C07281=1024.683,249.663,375.883,169.871,47.896,159.167
C07282=1024.672,249.258,375.931,169.865,47.901,159.167
C07283=1024.662,248.853,375.977,169.859,47.906,159.167
C07284=1024.652,248.448,376.024,169.852,47.911,159.167
C07285=1024.641,248.044,376.071,169.847,47.915,159.168
C07286=1024.635,247.795,376.099,169.843,47.919,159.168
C07287=1024.628,247.547,376.128,169.839,47.921,159.168
C07288=1024.622,247.299,376.157,169.835,47.924,159.168
C07289=1024.616,247.050,376.185,169.832,47.927,159.168
C07290=1024.609,246.802,376.213,169.827,47.930,159.168
C07291=1024.603,246.554,376.242,169.824,47.933,159.168
C07292=1024.597,246.305,376.271,169.821,47.935,159.168
C07293=1024.590,246.057,376.298,169.817,47.939,159.169
C07294=1024.584,245.809,376.327,169.813,47.941,159.169
C07295=1024.578,245.560,376.356,169.809,47.944,159.169
C07296=1024.572,245.312,376.385,169.806,47.947,159.169
C07297=1024.565,245.064,376.413,169.802,47.950,159.169
C07298=1024.560,244.816,376.441,169.799,47.953,159.169
C07299=1024.554,244.567,376.470,169.794,47.956,159.169
C07300=1024.547,244.320,376.498,169.791,47.959,159.170
C07301=1024.541,244.071,376.526,169.787,47.962,159.170
C07302=1024.535,243.823,376.555,169.784,47.965,159.170
C07303=1024.528,243.574,376.583,169.779,47.968,159.170
C07304=1024.522,243.325,376.611,169.776,47.971,159.170
C07305=1024.515,243.078,376.640,169.772,47.974,159.170
C07306=1024.508,242.829,376.668,169.769,47.977,159.170
C07307=1024.502,242.580,376.696,169.765,47.980,159.171
C07308=1024.495,242.333,376.724,169.762,47.983,159.171
C07309=1024.490,242.085,376.752,169.758,47.987,159.171
C07310=1024.483,241.836,376.780,169.754,47.989,159.171
C07311=1024.477,241.588,376.808,169.750,47.993,159.171
C07312=1024.471,241.339,376.836,169.747,47.996,159.171
C07313=1024.464,241.091,376.865,169.743,47.999,159.172
C07314=1024.458,240.842,376.893,169.740,48.002,159.172
C07315=1024.451,240.594,376.921,169.735,48.005,159.172
C07316=1024.445,240.345,376.949,169.732,48.008,159.172
C07317=1024.438,240.097,376.977,169.728,48.011,159.172
C07318=1024.432,239.850,377.005,169.725,48.015,159.173
C07319=1024.426,239.601,377.033,169.721,48.017,159.173
C07320=1024.419,239.352,377.061,169.718,48.020,159.173
C07321=1024.413,239.104,377.089,169.714,48.024,159.173
C07322=1024.406,238.856,377.116,169.711,48.027,159.173
C07323=1024.399,238.607,377.144,169.707,48.030,159.173
C07324=1024.394,238.359,377.172,169.703,48.033,159.174
C07325=1024.387,238.111,377.200,169.699,48.037,159.174
C07326=1024.381,237.862,377.227,169.696,48.040,159.174
C07327=1024.374,237.614,377.255,169.692,48.043,159.174
C07328=1024.367,237.365,377.283,169.688,48.047,159.174
C07329=1024.361,237.117,377.311,169.685,48.050,159.175
C07330=1024.355,236.869,377.339,169.681,48.053,159.175
C07331=1024.349,236.620,377.366,169.678,48.056,159.175
C07332=1024.342,236.372,377.394,169.674,48.060,159.175
C07333=1024.336,236.123,377.421,169.671,48.063,159.176
C07334=1024.329,235.874,377.449,169.667,48.066,159.176
C07335=1024.323,235.627,377.476,169.664,48.070,159.176
C07336=1024.316,235.378,377.504,169.660,48.073,159.176
C07337=1024.309,235.130,377.532,169.657,48.076,159.176
C07338=1024.299,234.719,377.577,169.650,48.082,159.177
C07339=1024.288,234.308,377.623,169.645,48.087,159.177
C07340=1024.277,233.897,377.668,169.638,48.093,159.177
C07341=1024.267,233.486,377.714,169.633,48.098,159.178
C07342=1024.260,233.238,377.741,169.629,48.101,159.178
C07343=1024.255,232.988,377.769,169.626,48.104,159.178
C07344=1024.248,232.740,377.797,169.622,48.108,159.179
C07345=1024.242,232.492,377.824,169.619,48.112,159.179
C07346=1024.235,232.244,377.852,169.615,48.115,159.179
C07347=1024.229,231.995,377.879,169.612,48.118,159.179
C07348=1024.223,231.747,377.906,169.608,48.122,159.179
C07349=1024.216,231.499,377.934,169.604,48.125,159.180
C07350=1024.210,231.249,377.961,169.600,48.128,159.180
C07351=1024.204,231.002,377.988,169.598,48.132,159.180
C07352=1024.197,230.753,378.016,169.594,48.135,159.180
C07353=1024.190,230.505,378.044,169.591,48.138,159.181
C07354=1024.185,230.256,378.071,169.586,48.142,159.181
C07355=1024.178,230.008,378.098,169.583,48.145,159.181
C07356=1024.172,229.759,378.125,169.580,48.149,159.181
C07357=1024.165,229.511,378.153,169.577,48.152,159.182
C07358=1024.159,229.262,378.180,169.573,48.156,159.182
C07359=1024.152,229.014,378.207,169.569,48.159,159.182
C07360=1024.146,228.766,378.235,169.566,48.163,159.182
C07361=1024.140,228.517,378.262,169.562,48.166,159.183
C07362=1024.133,228.268,378.289,169.559,48.169,159.183
C07363=1024.127,228.020,378.316,169.555,48.173,159.183
C07364=1024.120,227.772,378.343,169.552,48.177,159.183
C07365=1024.114,227.523,378.370,169.548,48.180,159.184
C07366=1024.108,227.275,378.398,169.545,48.184,159.184
C07367=1024.101,227.026,378.425,169.541,48.187,159.184
C07368=1024.095,226.778,378.451,169.538,48.190,159.184
C07369=1024.088,226.530,378.478,169.534,48.194,159.185
C07370=1024.082,226.281,378.505,169.531,48.198,159.185
C07371=1024.076,226.033,378.533,169.527,48.202,159.185
C07372=1024.068,225.784,378.559,169.524,48.205,159.186
C07373=1024.063,225.536,378.586,169.520,48.209,159.186
C07374=1024.056,225.287,378.614,169.516,48.212,159.186
C07375=1024.049,225.039,378.640,169.514,48.216,159.187
C07376=1024.043,224.790,378.667,169.510,48.220,159.187
C07377=1024.037,224.541,378.694,169.507,48.223,159.187
C07378=1024.031,224.293,378.721,169.503,48.227,159.187
C07379=1024.024,224.045,378.747,169.500,48.231,159.188
C07380=1024.018,223.796,378.774,169.496,48.234,159.188
C07381=1024.011,223.547,378.801,169.493,48.238,159.188
C07382=1024.004,223.299,378.828,169.489,48.241,159.189
C07383=1023.998,223.051,378.855,169.486,48.245,159.189
C07384=1023.992,222.802,378.882,169.482,48.248,159.189
C07385=1023.985,222.554,378.908,169.479,48.253,159.190
C07386=1023.979,222.305,378.936,169.476,48.256,159.190
C07387=1023.973,222.057,378.962,169.472,48.260,159.190
C07388=1023.966,221.808,378.989,169.469,48.263,159.190
C07389=1023.960,221.560,379.015,169.465,48.267,159.191
C07390=1023.954,221.311,379.042,169.462,48.271,159.191
C07391=1023.947,221.063,379.069,169.458,48.274,159.191
C07392=1023.940,220.814,379.096,169.456,48.278,159.192
C07393=1023.935,220.566,379.123,169.451,48.282,159.192
C07394=1023.924,220.147,379.168,169.446,48.288,159.192
C07395=1023.913,219.728,379.213,169.441,48.294,159.193
C07396=1023.902,219.309,379.258,169.434,48.301,159.194
C07397=1023.892,218.890,379.302,169.429,48.307,159.194
C07398=1023.885,218.641,379.329,169.426,48.311,159.195
C07399=1023.879,218.393,379.355,169.422,48.314,159.195
C07400=1023.872,218.144,379.382,169.419,48.318,159.195
C07401=1023.866,217.896,379.408,169.415,48.322,159.195
C07402=1023.859,217.648,379.434,169.412,48.326,159.196
C07403=1023.852,217.399,379.461,169.408,48.329,159.196
C07404=1023.847,217.151,379.487,169.406,48.333,159.196
C07405=1023.839,216.902,379.514,169.402,48.337,159.197
C07406=1023.834,216.654,379.540,169.398,48.342,159.197
C07407=1023.827,216.405,379.567,169.395,48.345,159.198
C07408=1023.820,216.157,379.593,169.392,48.349,159.198
C07409=1023.814,215.909,379.620,169.389,48.353,159.198
C07410=1023.808,215.659,379.645,169.385,48.357,159.199
C07411=1023.801,215.411,379.671,169.382,48.361,159.199
C07412=1023.795,215.162,379.698,169.378,48.365,159.199
C07413=1023.788,214.914,379.724,169.375,48.369,159.200
C07414=1023.782,214.666,379.751,169.372,48.373,159.200
C07415=1023.775,214.417,379.777,169.368,48.377,159.200
C07416=1023.769,214.168,379.803,169.365,48.380,159.201
C07417=1023.763,213.919,379.830,169.362,48.384,159.201
C07418=1023.756,213.671,379.856,169.359,48.388,159.201
C07419=1023.750,213.423,379.882,169.355,48.392,159.202
C07420=1023.743,213.174,379.909,169.351,48.396,159.202
C07421=1023.737,212.925,379.934,169.349,48.400,159.203
C07422=1023.731,212.677,379.960,169.345,48.404,159.203
C07423=1023.724,212.428,379.987,169.342,48.408,159.203
C07424=1023.718,212.180,380.013,169.338,48.412,159.204
C07425=1023.712,211.931,380.039,169.336,48.416,159.204
C07426=1023.705,211.682,380.066,169.332,48.420,159.204
C07427=1023.699,211.434,380.092,169.329,48.424,159.205
C07428=1023.693,211.185,380.118,169.326,48.428,159.205
C07429=1023.686,210.937,380.144,169.321,48.431,159.205
C07430=1023.679,210.689,380.170,169.319,48.435,159.206
C07431=1023.674,210.440,380.196,169.315,48.439,159.206
C07432=1023.667,210.192,380.222,169.312,48.443,159.207
C07433=1023.660,209.943,380.249,169.309,48.448,159.207
C07434=1023.654,209.694,380.274,169.306,48.452,159.208
C07435=1023.648,209.446,380.300,169.303,48.456,159.208
C07436=1023.642,209.196,380.326,169.299,48.460,159.208
C07437=1023.635,208.948,380.352,169.296,48.464,159.209
C07438=1023.629,208.700,380.378,169.292,48.468,159.209
C07439=1023.622,208.452,380.404,169.290,48.472,159.209
C07440=1023.615,208.203,380.430,169.286,48.476,159.210
C07441=1023.609,207.954,380.456,169.282,48.480,159.210
C07442=1023.603,207.706,380.482,169.279,48.484,159.211
C07443=1023.597,207.457,380.508,169.276,48.488,159.211
C07444=1023.590,207.208,380.534,169.273,48.492,159.212
C07445=1023.584,206.960,380.559,169.270,48.496,159.212
C07446=1023.577,206.712,380.585,169.266,48.501,159.212
C07447=1023.571,206.463,380.611,169.263,48.504,159.213
C07448=1023.564,206.214,380.636,169.260,48.509,159.213
C07449=1023.558,205.966,380.662,169.257,48.513,159.214
C07450=1023.547,205.550,380.705,169.251,48.520,159.214
C07451=1023.536,205.133,380.749,169.246,48.527,159.215
C07452=1023.525,204.716,380.791,169.240,48.534,159.216
C07453=1023.515,204.300,380.834,169.236,48.541,159.216
C07454=1023.491,203.269,380.934,168.819,48.442,159.136
C07455=1023.486,203.020,380.959,168.815,48.447,159.136
C07456=1023.480,202.772,380.983,168.811,48.452,159.136
C07457=1023.474,202.523,381.007,168.806,48.457,159.137
C07458=1023.469,202.274,381.031,168.802,48.463,159.137
C07459=1023.464,202.025,381.055,168.798,48.468,159.138
C07460=1023.458,201.776,381.079,168.794,48.472,159.138
C07461=1023.452,201.528,381.103,168.790,48.478,159.139
C07462=1023.446,201.279,381.127,168.786,48.483,159.139
C07463=1023.441,201.030,381.152,168.781,48.488,159.140
C07464=1023.436,200.781,381.175,168.778,48.493,159.140
C07465=1023.429,200.532,381.199,168.773,48.498,159.141
C07466=1023.424,200.284,381.223,168.769,48.503,159.141
C07467=1023.419,200.035,381.248,168.764,48.509,159.141
C07468=1023.413,199.786,381.272,168.761,48.513,159.142
C07469=1023.407,199.537,381.295,168.757,48.518,159.142
C07470=1023.402,199.288,381.319,168.753,48.524,159.143
C07471=1023.396,199.039,381.342,168.748,48.529,159.143
C07472=1023.390,198.791,381.366,168.744,48.534,159.144
C07473=1023.385,198.542,381.390,168.740,48.539,159.144
C07474=1023.378,198.293,381.414,168.736,48.545,159.145
C07475=1023.372,198.045,381.437,168.732,48.550,159.145
C07476=1023.367,197.795,381.461,168.727,48.555,159.146
C07477=1023.361,197.547,381.485,168.724,48.561,159.146
C07478=1023.356,197.298,381.508,168.720,48.566,159.147
C07479=1023.350,197.049,381.532,168.715,48.571,159.147
C07480=1023.344,196.800,381.555,168.711,48.576,159.148
C07481=1023.339,196.551,381.579,168.708,48.582,159.148
C07482=1023.333,196.303,381.602,168.703,48.587,159.149
C07483=1023.328,196.054,381.626,168.699,48.592,159.149
C07484=1023.322,195.805,381.649,168.695,48.598,159.150
C07485=1023.316,195.557,381.673,168.692,48.602,159.150
C07486=1023.310,195.307,381.697,168.687,48.608,159.151
C07487=1023.305,195.058,381.720,168.683,48.613,159.151
C07488=1023.299,194.810,381.744,168.679,48.619,159.152
C07489=1023.294,194.560,381.767,168.675,48.623,159.152
C07490=1023.288,194.312,381.791,168.671,48.628,159.152
C07491=1023.283,194.063,381.814,168.667,48.634,159.153
C07492=1023.277,193.814,381.837,168.663,48.639,159.154
C07493=1023.271,193.566,381.861,168.659,48.644,159.154
C07494=1023.266,193.317,381.884,168.655,48.650,159.155
C07495=1023.260,193.068,381.908,168.651,48.655,159.155
C07496=1023.254,192.819,381.931,168.647,48.660,159.155
C07497=1023.249,192.570,381.955,168.643,48.666,159.156
C07498=1023.243,192.321,381.978,168.640,48.671,159.157
C07499=1023.238,192.073,382.002,168.635,48.676,159.157
C07500=1023.232,191.824,382.025,168.631,48.682,159.158
C07501=1023.227,191.575,382.048,168.628,48.686,159.158
C07502=1023.221,191.326,382.072,168.623,48.692,159.158
C07503=1023.215,191.077,382.095,168.619,48.697,159.159
C07504=1023.210,190.829,382.118,168.616,48.702,159.160
C07505=1023.205,190.579,382.141,168.611,48.707,159.160
C07506=1023.199,190.331,382.165,168.607,48.713,159.161
C07507=1023.193,190.082,382.188,168.604,48.718,159.161
C07508=1023.188,189.833,382.212,168.600,48.724,159.162
C07509=1023.182,189.584,382.235,168.595,48.729,159.162
C07510=1023.177,189.336,382.259,168.592,48.734,159.163
C07511=1023.171,189.087,382.282,168.588,48.740,159.163
C07512=1023.166,188.838,382.305,168.584,48.744,159.164
C07513=1023.161,188.588,382.328,168.580,48.750,159.164
C07514=1023.155,188.340,382.351,168.576,48.755,159.165
C07515=1023.148,188.058,382.378,168.572,48.761,159.165
C07516=1023.142,187.776,382.404,168.568,48.767,159.166
C07517=1023.136,187.494,382.430,168.563,48.773,159.166
C07518=1023.131,187.212,382.457,168.559,48.779,159.167
C07519=1023.125,186.963,382.479,168.555,48.784,159.167
C07520=1023.119,186.714,382.502,168.551,48.790,159.168
C07521=1023.114,186.465,382.526,168.547,48.795,159.168
C07522=1023.108,186.216,382.549,168.543,48.800,159.169
C07523=1023.102,185.967,382.573,168.539,48.806,159.169
C07524=1023.097,185.718,382.596,168.536,48.810,159.170
C07525=1023.092,185.469,382.619,168.532,48.816,159.171
C07526=1023.087,185.221,382.642,168.529,48.821,159.171
C07527=1023.082,184.972,382.665,168.524,48.826,159.171
C07528=1023.076,184.723,382.688,168.521,48.832,159.172
C07529=1023.070,184.474,382.711,168.517,48.837,159.173
C07530=1023.065,184.225,382.735,168.513,48.842,159.173
C07531=1023.059,183.976,382.758,168.509,48.848,159.174
C07532=1023.054,183.728,382.780,168.506,48.853,159.174
C07533=1023.049,183.479,382.804,168.502,48.858,159.175
C07534=1023.044,183.230,382.827,168.498,48.863,159.175
C07535=1023.038,182.981,382.850,168.494,48.868,159.176
C07536=1023.033,182.731,382.872,168.491,48.874,159.176
C07537=1023.027,182.482,382.895,168.487,48.879,159.177
C07538=1023.022,182.234,382.918,168.484,48.885,159.177
C07539=1023.017,181.985,382.941,168.479,48.890,159.178
C07540=1023.011,181.735,382.963,168.475,48.896,159.178
C07541=1023.005,181.487,382.985,168.472,48.901,159.179
C07542=1022.999,181.238,383.008,168.468,48.907,159.180
C07543=1022.993,180.988,383.031,168.464,48.912,159.180
C07544=1022.988,180.741,383.053,168.461,48.918,159.181
C07545=1022.982,180.491,383.075,168.457,48.924,159.181
C07546=1022.976,180.242,383.098,168.453,48.929,159.182
C07547=1022.971,179.993,383.121,168.449,48.934,159.182
C07548=1022.965,179.744,383.142,168.445,48.940,159.183
C07549=1022.959,179.495,383.165,168.442,48.946,159.184
C07550=1022.954,179.246,383.187,168.438,48.951,159.184
C07551=1022.948,178.998,383.210,168.435,48.957,159.185
C07552=1022.942,178.748,383.232,168.431,48.962,159.185
C07553=1022.936,178.499,383.255,168.426,48.968,159.186
C07554=1022.931,178.251,383.276,168.423,48.973,159.186
C07555=1022.925,178.002,383.299,168.419,48.979,159.187
C07556=1022.920,177.752,383.321,168.416,48.985,159.188
C07557=1022.914,177.504,383.344,168.412,48.990,159.188
C07558=1022.908,177.255,383.365,168.409,48.995,159.189
C07559=1022.903,177.006,383.388,168.405,49.001,159.189
C07560=1022.897,176.757,383.411,168.401,49.006,159.190
C07561=1022.891,176.508,383.433,168.397,49.012,159.190
C07562=1022.886,176.259,383.455,168.393,49.018,159.191
C07563=1022.880,176.010,383.478,168.390,49.023,159.192
C07564=1022.874,175.761,383.499,168.386,49.029,159.192
C07565=1022.869,175.513,383.522,168.383,49.034,159.193
C07566=1022.863,175.263,383.544,168.379,49.040,159.193
C07567=1022.858,175.014,383.566,168.376,49.046,159.194
C07568=1022.852,174.766,383.588,168.371,49.051,159.194
C07569=1022.847,174.516,383.611,168.368,49.056,159.195
C07570=1022.841,174.268,383.634,168.364,49.062,159.195
C07571=1022.835,174.019,383.655,168.361,49.068,159.196
C07572=1022.830,173.770,383.677,168.357,49.073,159.197
C07573=1022.824,173.521,383.700,168.354,49.079,159.197
C07574=1022.819,173.272,383.721,168.350,49.084,159.198
C07575=1022.813,173.023,383.743,168.346,49.089,159.198
C07576=1022.808,172.774,383.766,168.342,49.095,159.199
C07577=1022.802,172.525,383.788,168.339,49.101,159.200
C07578=1022.797,172.276,383.810,168.335,49.107,159.200
C07579=1022.791,171.993,383.836,168.331,49.113,159.201
C07580=1022.784,171.711,383.860,168.328,49.119,159.201
C07581=1022.778,171.428,383.886,168.324,49.125,159.202
C07582=1022.771,171.146,383.911,168.320,49.132,159.203
C07583=1022.766,170.897,383.933,168.315,49.137,159.203
C07584=1022.760,170.648,383.954,168.312,49.142,159.204
C07585=1022.755,170.399,383.976,168.308,49.148,159.204
C07586=1022.750,170.150,383.999,168.305,49.154,159.205
C07587=1022.744,169.901,384.021,168.301,49.159,159.206
C07588=1022.739,169.652,384.042,168.298,49.165,159.206
C07589=1022.734,169.403,384.065,168.295,49.170,159.207
C07590=1022.728,169.154,384.086,168.291,49.176,159.207
C07591=1022.722,168.905,384.109,168.288,49.181,159.208
C07592=1022.717,168.657,384.131,168.284,49.187,159.208
C07593=1022.711,168.407,384.152,168.281,49.192,159.209
C07594=1022.706,168.158,384.175,168.277,49.197,159.210
C07595=1022.701,167.909,384.197,168.273,49.203,159.210
C07596=1022.695,167.660,384.218,168.270,49.209,159.211
C07597=1022.690,167.412,384.241,168.266,49.215,159.211
C07598=1022.684,167.162,384.263,168.263,49.220,159.212
C07599=1022.679,166.914,384.284,168.260,49.225,159.213
C07600=1022.674,166.665,384.306,168.256,49.231,159.213
C07601=1022.668,166.415,384.328,168.253,49.237,159.214
C07602=1022.663,166.167,384.350,168.250,49.242,159.214
C07603=1022.657,165.917,384.372,168.246,49.248,159.215
C07604=1022.653,165.669,384.394,168.243,49.253,159.216
C07605=1022.646,165.419,384.415,168.240,49.259,159.216
C07606=1022.642,165.170,384.437,168.235,49.264,159.217
C07607=1022.636,164.922,384.460,168.232,49.270,159.217
C07608=1022.630,164.673,384.481,168.228,49.276,159.218
C07609=1022.625,164.424,384.504,168.225,49.280,159.218
C07610=1022.620,164.175,384.525,168.222,49.286,159.219
C07611=1022.615,163.926,384.547,168.218,49.292,159.220
C07612=1022.609,163.677,384.569,168.215,49.298,159.220
C07613=1022.604,163.428,384.591,168.211,49.303,159.221
C07614=1022.598,163.179,384.612,168.209,49.308,159.221
C07615=1022.593,162.930,384.634,168.204,49.314,159.222
C07616=1022.588,162.681,384.656,168.201,49.319,159.222
C07617=1022.582,162.432,384.678,168.198,49.325,159.223
C07618=1022.578,162.183,384.700,168.194,49.331,159.224
C07619=1022.572,161.934,384.722,168.191,49.336,159.224
C07620=1022.567,161.684,384.743,168.188,49.341,159.225
C07621=1022.562,161.436,384.764,168.184,49.347,159.225
C07622=1022.556,161.186,384.786,168.181,49.353,159.226
C07623=1022.551,160.938,384.808,168.178,49.358,159.227
C07624=1022.546,160.689,384.830,168.175,49.363,159.227
C07625=1022.540,160.440,384.851,168.171,49.369,159.228
C07626=1022.535,160.191,384.873,168.168,49.375,159.228
C07627=1022.530,159.942,384.895,168.164,49.380,159.229
C07628=1022.524,159.693,384.917,168.161,49.385,159.230
C07629=1022.519,159.444,384.939,168.157,49.391,159.230
C07630=1022.515,159.194,384.960,168.154,49.397,159.231
C07631=1022.509,158.945,384.981,168.151,49.402,159.231
C07632=1022.503,158.697,385.003,168.147,49.408,159.232
C07633=1022.498,158.448,385.024,168.144,49.413,159.233
C07634=1022.492,158.198,385.045,168.141,49.419,159.233
C07635=1022.487,157.950,385.067,168.137,49.425,159.234
C07636=1022.482,157.700,385.087,168.134,49.431,159.234
C07637=1022.475,157.451,385.109,168.131,49.436,159.235
C07638=1022.470,157.203,385.130,168.127,49.442,159.236
C07639=1022.465,156.953,385.151,168.124,49.448,159.236
C07640=1022.459,156.704,385.173,168.121,49.453,159.237
C07641=1022.454,156.456,385.194,168.117,49.459,159.238
C07642=1022.448,156.207,385.215,168.114,49.465,159.238
C07643=1022.442,155.924,385.239,168.110,49.471,159.239
C07644=1022.436,155.640,385.263,168.106,49.477,159.240
C07645=1022.429,155.358,385.287,168.103,49.484,159.240
C07646=1022.423,155.075,385.311,168.099,49.491,159.241
C07647=1022.418,154.826,385.332,168.096,49.496,159.242
C07648=1022.413,154.577,385.354,168.092,49.502,159.242
C07649=1022.407,154.327,385.375,168.089,49.507,159.243
C07650=1022.402,154.079,385.396,168.086,49.513,159.243
C07651=1022.396,153.830,385.417,168.082,49.519,159.244
C07652=1022.390,153.580,385.438,168.079,49.525,159.245
C07653=1022.385,153.331,385.459,168.076,49.530,159.245
C07654=1022.380,153.083,385.481,168.073,49.536,159.246
C07655=1022.375,152.833,385.501,168.069,49.542,159.247
C07656=1022.369,152.584,385.522,168.066,49.547,159.247
C07657=1022.363,152.335,385.543,168.063,49.553,159.248
C07658=1022.358,152.086,385.564,168.059,49.559,159.249
C07659=1022.353,151.837,385.585,168.056,49.565,159.249
C07660=1022.347,151.588,385.606,168.053,49.570,159.250
C07661=1022.341,151.338,385.627,168.049,49.576,159.250
C07662=1022.336,151.090,385.648,168.046,49.582,159.251
C07663=1022.331,150.841,385.669,168.043,49.588,159.252
C07664=1022.325,150.592,385.689,168.040,49.593,159.252
C07665=1022.319,150.343,385.711,168.036,49.599,159.253
C07666=1022.314,150.093,385.731,168.034,49.605,159.254
C07667=1022.309,149.844,385.752,168.031,49.611,159.254
C07668=1022.303,149.596,385.773,168.028,49.616,159.255
C07669=1022.298,149.347,385.794,168.024,49.622,159.256
C07670=1022.292,149.097,385.815,168.021,49.628,159.256
C07671=1022.286,148.848,385.836,168.018,49.633,159.257
C07672=1022.281,148.599,385.856,168.014,49.639,159.257
C07673=1022.276,148.350,385.877,168.011,49.645,159.258
C07674=1022.271,148.101,385.897,168.008,49.651,159.259
C07675=1022.265,147.852,385.919,168.005,49.656,159.259
C07676=1022.259,147.603,385.940,168.001,49.662,159.260
C07677=1022.254,147.353,385.960,167.998,49.668,159.261
C07678=1022.249,147.104,385.981,167.995,49.674,159.261
C07679=1022.243,146.856,386.002,167.992,49.679,159.262
C07680=1022.238,146.607,386.023,167.988,49.685,159.263
C07681=1022.232,146.358,386.043,167.985,49.691,159.263
C07682=1022.226,146.108,386.063,167.982,49.697,159.264
C07683=1022.221,145.859,386.084,167.979,49.702,159.265
C07684=1022.216,145.610,386.105,167.975,49.708,159.265
C07685=1022.210,145.361,386.125,167.972,49.714,159.266
C07686=1022.205,145.112,386.146,167.970,49.720,159.267
C07687=1022.199,144.863,386.166,167.967,49.726,159.267
C07688=1022.194,144.614,386.187,167.963,49.732,159.268
C07689=1022.188,144.364,386.208,167.960,49.738,159.268
C07690=1022.182,144.115,386.228,167.957,49.743,159.269
C07691=1022.176,143.867,386.248,167.954,49.749,159.270
C07692=1022.171,143.617,386.269,167.950,49.755,159.270
C07693=1022.166,143.368,386.289,167.947,49.761,159.271
C07694=1022.161,143.119,386.310,167.944,49.766,159.272
C07695=1022.155,142.870,386.330,167.941,49.772,159.272
C07696=1022.149,142.621,386.351,167.937,49.778,159.273
C07697=1022.144,142.372,386.371,167.935,49.784,159.274
C07698=1022.138,142.123,386.391,167.932,49.790,159.274
C07699=1022.133,141.874,386.412,167.929,49.796,159.275
C07700=1022.127,141.624,386.433,167.926,49.801,159.276
C07701=1022.122,141.375,386.453,167.922,49.807,159.276
C07702=1022.116,141.126,386.473,167.919,49.813,159.277
C07703=1022.111,140.877,386.494,167.916,49.819,159.278
C07704=1022.105,140.628,386.514,167.913,49.825,159.278
C07705=1022.100,140.379,386.535,167.909,49.831,159.279
C07706=1022.094,140.130,386.554,167.906,49.836,159.280
C07707=1022.089,139.893,386.574,167.904,49.842,159.280
C07708=1022.084,139.654,386.593,167.901,49.848,159.281
C07709=1022.079,139.416,386.613,167.898,49.853,159.282
C07710=1022.074,139.177,386.632,167.894,49.858,159.282
C07711=1022.069,138.940,386.652,167.891,49.864,159.283
C07712=1022.064,138.701,386.671,167.890,49.869,159.283
C07713=1022.058,138.463,386.691,167.887,49.875,159.284
C07714=1022.053,138.225,386.709,167.884,49.881,159.285
C07715=1022.047,137.919,386.735,167.879,49.888,159.285
C07716=1022.040,137.615,386.760,167.876,49.895,159.286
C07717=1022.033,137.310,386.784,167.871,49.902,159.287
C07718=1022.026,137.004,386.809,167.868,49.910,159.288
C07719=1022.020,136.755,386.829,167.865,49.915,159.289
C07720=1022.015,136.506,386.849,167.862,49.921,159.289
C07721=1022.009,136.257,386.869,167.859,49.927,159.290
C07722=1022.004,136.007,386.889,167.855,49.933,159.290
C07723=1021.998,135.759,386.909,167.853,49.938,159.291
C07724=1021.993,135.509,386.929,167.850,49.944,159.292
C07725=1021.987,135.260,386.949,167.847,49.950,159.293
C07726=1021.982,135.012,386.969,167.844,49.956,159.293
C07727=1021.977,134.762,386.988,167.840,49.962,159.294
C07728=1021.971,134.513,387.009,167.837,49.968,159.295
C07729=1021.965,134.264,387.029,167.834,49.974,159.295
C07730=1021.960,134.015,387.049,167.831,49.979,159.296
C07731=1021.954,133.766,387.069,167.829,49.985,159.296
C07732=1021.949,133.517,387.089,167.825,49.992,159.297
C07733=1021.943,133.267,387.108,167.822,49.997,159.298
C07734=1021.938,133.018,387.129,167.819,50.003,159.299
C07735=1021.932,132.769,387.149,167.816,50.009,159.299
C07736=1021.927,132.519,387.169,167.813,50.015,159.300
C07737=1021.921,132.271,387.189,167.810,50.020,159.301
C07738=1021.916,132.021,387.208,167.807,50.026,159.301
C07739=1021.910,131.772,387.228,167.804,50.033,159.302
C07740=1021.905,131.524,387.248,167.801,50.038,159.303
C07741=1021.900,131.274,387.268,167.798,50.044,159.303
C07742=1021.894,131.025,387.288,167.795,50.050,159.304
C07743=1021.889,130.776,387.308,167.792,50.056,159.305
C07744=1021.883,130.527,387.328,167.790,50.061,159.305
C07745=1021.878,130.277,387.347,167.786,50.067,159.306
C07746=1021.872,130.028,387.367,167.783,50.073,159.306
C07747=1021.866,129.779,387.387,167.780,50.079,159.307
C07748=1021.861,129.530,387.407,167.777,50.085,159.308
C07749=1021.856,129.281,387.426,167.774,50.091,159.309
C07750=1021.850,129.032,387.445,167.771,50.098,159.309
C07751=1021.844,128.783,387.465,167.768,50.103,159.310
C07752=1021.839,128.533,387.485,167.765,50.109,159.311
C07753=1021.833,128.284,387.504,167.762,50.115,159.311
C07754=1021.827,128.035,387.524,167.760,50.121,159.312
C07755=1021.821,127.786,387.543,167.756,50.127,159.313
C07756=1021.816,127.536,387.563,167.753,50.133,159.313
C07757=1021.810,127.287,387.583,167.750,50.139,159.314
C07758=1021.805,127.038,387.602,167.747,50.145,159.315
C07759=1021.800,126.789,387.621,167.745,50.151,159.316
C07760=1021.794,126.540,387.641,167.741,50.157,159.316
C07761=1021.788,126.291,387.660,167.738,50.163,159.317
C07762=1021.782,126.041,387.679,167.735,50.169,159.318
C07763=1021.776,125.792,387.699,167.732,50.175,159.318
C07764=1021.771,125.544,387.718,167.729,50.181,159.319
C07765=1021.766,125.294,387.738,167.726,50.187,159.320
C07766=1021.761,125.045,387.757,167.723,50.193,159.320
C07767=1021.755,124.796,387.777,167.720,50.199,159.321
C07768=1021.749,124.546,387.796,167.717,50.205,159.322
C07769=1021.744,124.298,387.815,167.715,50.211,159.323
C07770=1021.738,124.048,387.835,167.712,50.217,159.323
C07771=1021.732,123.765,387.857,167.708,50.223,159.324
C07772=1021.726,123.482,387.879,167.705,50.230,159.325
C07773=1021.719,123.198,387.901,167.701,50.237,159.325
C07774=1021.713,122.915,387.923,167.698,50.244,159.326
C07775=1021.707,122.666,387.942,167.695,50.249,159.327
C07776=1021.701,122.417,387.962,167.692,50.256,159.328
C07777=1021.696,122.168,387.981,167.690,50.262,159.328
C07778=1021.691,121.919,388.000,167.687,50.267,159.329
C07779=1021.685,121.669,388.020,167.684,50.273,159.330
C07780=1021.679,121.420,388.039,167.681,50.279,159.330
C07781=1021.674,121.171,388.058,167.677,50.286,159.331
C07782=1021.668,120.922,388.078,167.675,50.291,159.332
C07783=1021.662,120.673,388.097,167.672,50.297,159.332
C07784=1021.658,120.424,388.117,167.669,50.303,159.333
C07785=1021.652,120.174,388.136,167.666,50.309,159.334
C07786=1021.647,119.925,388.155,167.663,50.315,159.335
C07787=1021.641,119.675,388.174,167.661,50.321,159.335
C07788=1021.636,119.427,388.193,167.658,50.327,159.336
C07789=1021.630,119.177,388.212,167.655,50.332,159.337
C07790=1021.624,118.928,388.232,167.652,50.338,159.337
C07791=1021.619,118.680,388.251,167.648,50.344,159.338
C07792=1021.614,118.430,388.270,167.646,50.351,159.339
C07793=1021.608,118.181,388.290,167.643,50.356,159.339
C07794=1021.603,117.931,388.310,167.640,50.362,159.340
C07795=1021.598,117.682,388.328,167.637,50.368,159.341
C07796=1021.592,117.433,388.348,167.634,50.374,159.341
C07797=1021.586,117.183,388.367,167.631,50.379,159.342
C07798=1021.581,116.935,388.386,167.629,50.386,159.343
C07799=1021.576,116.685,388.405,167.626,50.392,159.343
C07800=1021.570,116.436,388.424,167.623,50.397,159.344
C07801=1021.565,116.187,388.443,167.620,50.403,159.345
C07802=1021.559,115.938,388.462,167.617,50.409,159.345
C07803=1021.554,115.689,388.481,167.615,50.415,159.346
C07804=1021.548,115.440,388.501,167.612,50.421,159.347
C07805=1021.543,115.190,388.520,167.609,50.426,159.347
C07806=1021.538,114.941,388.539,167.606,50.433,159.348
C07807=1021.533,114.692,388.558,167.604,50.439,159.349
C07808=1021.527,114.442,388.578,167.601,50.444,159.349
C07809=1021.522,114.193,388.597,167.598,50.450,159.350
C07810=1021.516,113.944,388.616,167.595,50.456,159.351
C07811=1021.511,113.695,388.635,167.592,50.462,159.351
C07812=1021.505,113.446,388.654,167.588,50.468,159.352
C07813=1021.500,113.196,388.673,167.585,50.474,159.353
C07814=1021.495,112.948,388.692,167.583,50.479,159.353
C07815=1021.489,112.698,388.711,167.580,50.485,159.354
C07816=1021.483,112.449,388.731,167.577,50.492,159.355
C07817=1021.479,112.200,388.749,167.574,50.497,159.355
C07818=1021.473,111.950,388.768,167.572,50.503,159.356
C07819=1021.468,111.701,388.787,167.569,50.509,159.357
C07820=1021.462,111.452,388.806,167.566,50.515,159.357
C07821=1021.456,111.203,388.825,167.563,50.521,159.358
C07822=1021.451,110.953,388.843,167.561,50.527,159.359
C07823=1021.445,110.704,388.862,167.558,50.533,159.360
C07824=1021.440,110.455,388.881,167.555,50.539,159.360
C07825=1021.434,110.206,388.900,167.552,50.545,159.361
C07826=1021.428,109.956,388.918,167.550,50.551,159.362
C07827=1021.423,109.707,388.937,167.547,50.557,159.362
C07828=1021.417,109.458,388.956,167.544,50.562,159.363
C07829=1021.412,109.209,388.974,167.540,50.569,159.364
C07830=1021.406,108.959,388.993,167.538,50.575,159.364
C07831=1021.401,108.711,389.012,167.535,50.581,159.365
C07832=1021.395,108.461,389.030,167.532,50.587,159.366
C07833=1021.389,108.212,389.049,167.529,50.593,159.367
C07834=1021.385,107.962,389.067,167.527,50.599,159.367
C07835=1021.378,107.680,389.089,167.523,50.606,159.368
C07836=1021.372,107.396,389.109,167.520,50.612,159.369
C07837=1021.365,107.112,389.130,167.517,50.619,159.370
C07838=1021.359,106.829,389.152,167.514,50.626,159.371
C07839=1021.353,106.580,389.170,167.511,50.632,159.371
C07840=1021.347,106.331,389.189,167.509,50.638,159.372
C07841=1021.343,106.082,389.207,167.506,50.644,159.373
C07842=1021.336,105.832,389.226,167.503,50.650,159.373
C07843=1021.331,105.584,389.245,167.499,50.656,159.374
C07844=1021.325,105.334,389.263,167.497,50.662,159.375
C07845=1021.320,105.085,389.282,167.494,50.668,159.375
C07846=1021.315,104.835,389.300,167.491,50.675,159.376
C07847=1021.309,104.587,389.318,167.488,50.680,159.377
C07848=1021.303,104.337,389.337,167.486,50.686,159.377
C07849=1021.297,104.088,389.355,167.483,50.692,159.378
C07850=1021.292,103.838,389.374,167.480,50.698,159.379
C07851=1021.287,103.590,389.393,167.478,50.704,159.380
C07852=1021.281,103.340,389.411,167.475,50.710,159.380
C07853=1021.276,103.091,389.429,167.472,50.716,159.381
C07854=1021.270,102.841,389.447,167.469,50.722,159.382
C07855=1021.265,102.593,389.466,167.467,50.728,159.382
C07856=1021.259,102.343,389.485,167.464,50.734,159.383
C07857=1021.253,102.094,389.503,167.461,50.740,159.384
C07858=1021.248,101.844,389.522,167.458,50.746,159.384
C07859=1021.242,101.595,389.539,167.455,50.751,159.385
C07860=1021.237,101.346,389.558,167.453,50.758,159.386
C07861=1021.232,101.096,389.577,167.450,50.764,159.386
C07862=1021.226,100.848,389.595,167.447,50.770,159.387
C07863=1021.221,100.598,389.613,167.445,50.775,159.388
C07864=1021.215,100.349,389.632,167.442,50.781,159.388
C07865=1021.210,100.099,389.650,167.439,50.787,159.389
C07866=1021.204,99.850,389.668,167.437,50.794,159.390
C07867=1021.198,99.601,389.687,167.434,50.799,159.391
C07868=1021.194,99.351,389.705,167.431,50.805,159.391
C07869=1021.188,99.102,389.723,167.428,50.811,159.392
C07870=1021.182,98.853,389.741,167.426,50.818,159.393
C07871=1021.177,98.604,389.760,167.423,50.823,159.393
C07872=1021.171,98.354,389.777,167.420,50.829,159.394
C07873=1021.165,98.105,389.795,167.416,50.835,159.395
C07874=1021.160,97.856,389.814,167.414,50.842,159.395
C07875=1021.154,97.607,389.832,167.411,50.848,159.396
C07876=1021.149,97.358,389.849,167.408,50.854,159.397
C07877=1021.142,97.108,389.867,167.406,50.860,159.398
C07878=1021.137,96.859,389.886,167.403,50.866,159.398
C07879=1021.131,96.609,389.904,167.400,50.872,159.399
C07880=1021.126,96.360,389.922,167.397,50.878,159.400
C07881=1021.121,96.111,389.940,167.395,50.884,159.400
C07882=1021.115,95.861,389.958,167.392,50.890,159.401
C07883=1021.109,95.613,389.976,167.389,50.896,159.402
C07884=1021.104,95.363,389.995,167.387,50.902,159.402
C07885=1021.098,95.114,390.012,167.384,50.908,159.403
C07886=1021.093,94.865,390.030,167.381,50.914,159.404
C07887=1021.086,94.615,390.048,167.379,50.920,159.405
C07888=1021.082,94.366,390.066,167.376,50.926,159.405
C07889=1021.076,94.117,390.084,167.374,50.932,159.406
C07890=1021.070,93.868,390.102,167.371,50.938,159.407
C07891=1021.065,93.618,390.120,167.368,50.944,159.407
C07892=1021.059,93.369,390.138,167.365,50.950,159.408
C07893=1021.053,93.119,390.156,167.363,50.956,159.409
C07894=1021.048,92.870,390.173,167.360,50.962,159.410
C07895=1021.043,92.621,390.191,167.357,50.968,159.410
C07896=1021.037,92.371,390.209,167.354,50.974,159.411
C07897=1021.031,92.122,390.227,167.352,50.980,159.411
C07898=1021.026,91.873,390.246,167.349,50.986,159.412
C07899=1021.019,91.590,390.265,167.346,50.993,159.413
C07900=1021.013,91.307,390.286,167.342,51.000,159.414
C07901=1021.007,91.023,390.306,167.340,51.006,159.415
C07902=1021.001,90.741,390.327,167.337,51.013,159.415
C07903=1020.995,90.491,390.345,167.334,51.019,159.416
C07904=1020.990,90.242,390.363,167.331,51.025,159.417
C07905=1020.984,89.993,390.380,167.328,51.031,159.417
C07906=1020.979,89.744,390.398,167.325,51.037,159.418
C07907=1020.974,89.494,390.417,167.323,51.043,159.419
C07908=1020.968,89.245,390.434,167.320,51.049,159.420
C07909=1020.963,88.996,390.452,167.318,51.055,159.420
C07910=1020.956,88.746,390.470,167.315,51.061,159.421
C07911=1020.951,88.497,390.487,167.312,51.067,159.421
C07912=1020.946,88.247,390.504,167.310,51.073,159.422
C07913=1020.940,87.997,390.522,167.307,51.079,159.423
C07914=1020.934,87.748,390.540,167.304,51.085,159.424
C07915=1020.929,87.499,390.557,167.302,51.092,159.424
C07916=1020.923,87.250,390.575,167.299,51.097,159.425
C07917=1020.917,87.001,390.593,167.296,51.103,159.426
C07918=1020.911,86.751,390.610,167.294,51.110,159.427
C07919=1020.906,86.502,390.627,167.291,51.116,159.427
C07920=1020.901,86.253,390.645,167.288,51.122,159.428
C07921=1020.895,86.003,390.663,167.285,51.127,159.429
C07922=1020.889,85.754,390.680,167.282,51.134,159.429
C07923=1020.883,85.505,390.698,167.279,51.140,159.430
C07924=1020.878,85.255,390.714,167.277,51.146,159.431
C07925=1020.872,85.006,390.732,167.274,51.152,159.431
C07926=1020.867,84.757,390.750,167.271,51.158,159.432
C07927=1020.861,84.507,390.768,167.269,51.164,159.433
C07928=1020.856,84.258,390.785,167.266,51.170,159.433
C07929=1020.849,84.008,390.802,167.263,51.176,159.434
C07930=1020.844,83.759,390.819,167.261,51.183,159.435
C07931=1020.838,83.510,390.837,167.258,51.189,159.436
C07932=1020.832,83.261,390.854,167.255,51.194,159.436
C07933=1020.827,83.012,390.871,167.253,51.200,159.437
C07934=1020.821,82.762,390.889,167.250,51.206,159.438
C07935=1020.816,82.513,390.907,167.247,51.213,159.438
C07936=1020.810,82.264,390.924,167.245,51.219,159.439
C07937=1020.805,82.014,390.941,167.242,51.224,159.440
C07938=1020.799,81.765,390.959,167.239,51.230,159.440
C07939=1020.794,81.516,390.976,167.236,51.236,159.441
C07940=1020.788,81.266,390.994,167.234,51.243,159.442
C07941=1020.783,81.017,391.011,167.231,51.249,159.443
C07942=1020.777,80.768,391.029,167.229,51.255,159.443
C07943=1020.772,80.518,391.046,167.226,51.260,159.444
C07944=1020.766,80.269,391.063,167.223,51.266,159.444
C07945=1020.761,80.020,391.081,167.221,51.272,159.445
C07946=1020.755,79.770,391.099,167.219,51.278,159.446
C07947=1020.749,79.520,391.115,167.216,51.284,159.447
C07948=1020.744,79.271,391.133,167.213,51.290,159.447
C07949=1020.739,79.022,391.150,167.211,51.296,159.448
C07950=1020.733,78.773,391.167,167.208,51.302,159.449
C07951=1020.728,78.524,391.185,167.205,51.308,159.449
C07952=1020.722,78.274,391.202,167.202,51.314,159.450
C07953=1020.717,78.025,391.219,167.200,51.320,159.451
C07954=1020.711,77.775,391.237,167.197,51.326,159.451
C07955=1020.706,77.526,391.254,167.195,51.332,159.452
C07956=1020.699,77.277,391.271,167.192,51.338,159.453
C07957=1020.694,77.027,391.288,167.189,51.344,159.453
C07958=1020.689,76.778,391.306,167.186,51.350,159.454
C07959=1020.683,76.528,391.322,167.184,51.356,159.455
C07960=1020.678,76.279,391.340,167.181,51.362,159.456
C07961=1020.672,76.030,391.356,167.179,51.368,159.456
C07962=1020.666,75.781,391.374,167.176,51.374,159.457
C07963=1020.660,75.498,391.393,167.173,51.381,159.458
C07964=1020.653,75.215,391.412,167.170,51.388,159.458
C07965=1020.647,74.931,391.432,167.167,51.395,159.459
C07966=1020.641,74.648,391.451,167.164,51.402,159.460
C07967=1020.635,74.399,391.468,167.161,51.407,159.461
C07968=1020.630,74.150,391.485,167.158,51.414,159.461
C07969=1020.624,73.900,391.502,167.156,51.420,159.462
C07970=1020.618,73.651,391.519,167.153,51.426,159.463
C07971=1020.612,73.401,391.536,167.150,51.432,159.463
C07972=1020.607,73.152,391.553,167.148,51.438,159.464
C07973=1020.601,72.902,391.570,167.145,51.444,159.465
C07974=1020.596,72.653,391.587,167.142,51.450,159.466
C07975=1020.590,72.404,391.604,167.140,51.456,159.466
C07976=1020.584,72.154,391.620,167.137,51.462,159.467
C07977=1020.579,71.905,391.638,167.134,51.468,159.468
C07978=1020.573,71.656,391.655,167.132,51.474,159.468
C07979=1020.568,71.406,391.671,167.129,51.480,159.469
C07980=1020.562,71.157,391.689,167.127,51.486,159.470
C07981=1020.557,70.908,391.706,167.124,51.492,159.470
C07982=1020.551,70.658,391.722,167.121,51.498,159.471
C07983=1020.546,70.409,391.739,167.118,51.504,159.472
C07984=1020.539,70.160,391.756,167.116,51.510,159.472
C07985=1020.534,69.910,391.772,167.114,51.516,159.473
C07986=1020.529,69.661,391.789,167.112,51.522,159.474
C07987=1020.523,69.412,391.806,167.109,51.528,159.475
C07988=1020.517,69.162,391.823,167.106,51.534,159.475
C07989=1020.512,68.913,391.840,167.104,51.540,159.476
C07990=1020.506,68.663,391.856,167.101,51.546,159.476
C07991=1020.501,68.414,391.874,167.098,51.552,159.477
C07992=1020.495,68.165,391.890,167.095,51.558,159.478
C07993=1020.490,67.915,391.907,167.093,51.564,159.479
C07994=1020.484,67.666,391.923,167.090,51.570,159.479
C07995=1020.478,67.416,391.940,167.088,51.576,159.480
C07996=1020.472,67.167,391.957,167.085,51.582,159.481
C07997=1020.467,66.918,391.974,167.082,51.588,159.481
C07998=1020.461,66.668,391.990,167.080,51.594,159.482
C07999=1020.456,66.419,392.007,167.077,51.601,159.483
C08000=1020.450,66.169,392.023,167.075,51.606,159.483
C08001=1020.445,65.920,392.040,167.072,51.612,159.484
C08002=1020.439,65.670,392.056,167.069,51.618,159.485
C08003=1020.433,65.421,392.074,167.066,51.624,159.485
C08004=1020.427,65.172,392.090,167.064,51.630,159.486
C08005=1020.421,64.923,392.106,167.061,51.637,159.487
C08006=1020.416,64.673,392.123,167.059,51.643,159.487
C08007=1020.410,64.424,392.139,167.056,51.649,159.488
C08008=1020.406,64.175,392.156,167.053,51.655,159.489
C08009=1020.400,63.925,392.172,167.051,51.661,159.489
C08010=1020.394,63.676,392.189,167.048,51.666,159.490
C08011=1020.388,63.426,392.205,167.045,51.672,159.491
C08012=1020.382,63.177,392.222,167.043,51.678,159.491
C08013=1020.377,62.927,392.238,167.040,51.685,159.492
C08014=1020.371,62.678,392.255,167.038,51.691,159.493
C08015=1020.365,62.429,392.271,167.035,51.697,159.494
C08016=1020.359,62.179,392.287,167.033,51.703,159.494
C08017=1020.353,61.930,392.303,167.030,51.709,159.495
C08018=1020.348,61.680,392.320,167.027,51.715,159.496
C08019=1020.343,61.430,392.336,167.025,51.721,159.496
C08020=1020.337,61.181,392.352,167.022,51.728,159.497
C08021=1020.331,60.932,392.368,167.019,51.734,159.498
C08022=1020.325,60.682,392.385,167.016,51.740,159.498
C08023=1020.319,60.434,392.401,167.013,51.746,159.499
C08024=1020.313,60.184,392.417,167.011,51.753,159.500
C08025=1020.307,59.935,392.433,167.008,51.759,159.501
C08026=1020.303,59.685,392.449,167.005,51.765,159.501
C08027=1020.296,59.402,392.468,167.003,51.771,159.502
C08028=1020.289,59.118,392.486,167.000,51.778,159.503
C08029=1020.282,58.835,392.505,166.997,51.785,159.503
C08030=1020.276,58.552,392.523,166.993,51.792,159.504
C08031=1020.270,58.302,392.539,166.991,51.799,159.505
C08032=1020.264,58.053,392.555,166.988,51.805,159.506
C08033=1020.259,57.803,392.571,166.986,51.811,159.506
C08034=1020.253,57.555,392.587,166.983,51.817,159.507
C08035=1020.247,57.305,392.603,166.980,51.823,159.508
C08036=1020.241,57.056,392.619,166.978,51.829,159.509
C08037=1020.236,56.806,392.635,166.975,51.835,159.509
C08038=1020.231,56.556,392.652,166.973,51.841,159.510
C08039=1020.225,56.307,392.668,166.970,51.847,159.510
C08040=1020.219,56.058,392.684,166.967,51.853,159.511
C08041=1020.214,55.808,392.699,166.965,51.859,159.512
C08042=1020.208,55.559,392.716,166.962,51.866,159.513
C08043=1020.202,55.310,392.732,166.960,51.872,159.513
C08044=1020.196,55.060,392.748,166.957,51.878,159.514
C08045=1020.191,54.811,392.763,166.954,51.884,159.515
C08046=1020.185,54.562,392.780,166.952,51.890,159.515
C08047=1020.179,54.312,392.796,166.949,51.896,159.516
C08048=1020.174,54.063,392.813,166.946,51.902,159.516
C08049=1020.168,53.813,392.828,166.944,51.908,159.517
C08050=1020.163,53.564,392.844,166.941,51.914,159.518
C08051=1020.157,53.315,392.860,166.939,51.920,159.519
C08052=1020.151,53.065,392.876,166.936,51.926,159.519
C08053=1020.145,52.815,392.892,166.933,51.932,159.520
C08054=1020.139,52.566,392.908,166.931,51.938,159.521
C08055=1020.134,52.317,392.924,166.928,51.944,159.521
C08056=1020.128,52.067,392.940,166.926,51.950,159.522
C08057=1020.122,51.818,392.956,166.923,51.956,159.523
C08058=1020.117,51.568,392.972,166.920,51.962,159.523
C08059=1020.112,51.319,392.988,166.918,51.968,159.524
C08060=1020.106,51.069,393.004,166.915,51.974,159.524
C08061=1020.100,50.820,393.020,166.912,51.980,159.525
C08062=1020.095,50.571,393.036,166.910,51.986,159.526
C08063=1020.089,50.321,393.051,166.908,51.992,159.527
C08064=1020.083,50.072,393.068,166.905,51.998,159.527
C08065=1020.077,49.822,393.084,166.903,52.004,159.528
C08066=1020.072,49.573,393.099,166.900,52.010,159.528
C08067=1020.066,49.324,393.115,166.897,52.015,159.529
C08068=1020.061,49.074,393.131,166.895,52.021,159.530
C08069=1020.056,48.825,393.147,166.892,52.027,159.530
C08070=1020.051,48.575,393.163,166.889,52.033,159.531
C08071=1020.045,48.326,393.179,166.887,52.039,159.532
C08072=1020.039,48.076,393.195,166.884,52.045,159.532
C08073=1020.034,47.827,393.211,166.881,52.051,159.533
C08074=1020.028,47.578,393.227,166.879,52.057,159.534
C08075=1020.022,47.328,393.242,166.876,52.063,159.534
C08076=1020.017,47.079,393.258,166.873,52.069,159.535
C08077=1020.011,46.829,393.274,166.871,52.075,159.536
C08078=1020.005,46.580,393.290,166.869,52.081,159.536
C08079=1020.000,46.330,393.305,166.867,52.087,159.537
C08080=1019.994,46.081,393.321,166.863,52.092,159.537
C08081=1019.989,45.831,393.338,166.861,52.098,159.538
C08082=1019.984,45.582,393.353,166.858,52.104,159.539
C08083=1019.978,45.332,393.369,166.856,52.110,159.539
C08084=1019.973,45.084,393.385,166.853,52.116,159.540
C08085=1019.967,44.834,393.400,166.850,52.122,159.541
C08086=1019.961,44.584,393.417,166.848,52.128,159.541
C08087=1019.956,44.335,393.432,166.845,52.134,159.542
C08088=1019.950,44.086,393.448,166.842,52.140,159.543
C08089=1019.945,43.836,393.464,166.840,52.145,159.543
C08090=1019.939,43.587,393.480,166.838,52.151,159.544
C08091=1019.934,43.303,393.497,166.834,52.158,159.545
C08092=1019.927,43.020,393.515,166.832,52.164,159.545
C08093=1019.921,42.736,393.533,166.829,52.171,159.546
C08094=1019.914,42.453,393.551,166.826,52.178,159.547
C08095=1019.909,42.203,393.566,166.824,52.184,159.547
C08096=1019.903,41.954,393.582,166.821,52.190,159.548
C08097=1019.898,41.704,393.598,166.818,52.196,159.549
C08098=1019.892,41.454,393.613,166.816,52.202,159.549
C08099=1019.886,41.206,393.629,166.813,52.208,159.550
C08100=1019.880,40.956,393.644,166.811,52.214,159.551
C08101=1019.875,40.707,393.659,166.808,52.220,159.551
C08102=1019.870,40.457,393.675,166.805,52.226,159.552
C08103=1019.863,40.208,393.690,166.803,52.232,159.553
C08104=1019.858,39.959,393.706,166.800,52.237,159.553
C08105=1019.852,39.709,393.721,166.797,52.243,159.554
C08106=1019.847,39.459,393.736,166.794,52.249,159.554
C08107=1019.842,39.209,393.752,166.792,52.255,159.555
C08108=1019.836,38.961,393.767,166.789,52.261,159.556
C08109=1019.830,38.711,393.783,166.786,52.267,159.556
C08110=1019.825,38.462,393.798,166.784,52.273,159.557
C08111=1019.819,38.212,393.813,166.781,52.279,159.557
C08112=1019.813,37.963,393.830,166.779,52.285,159.558
C08113=1019.807,37.714,393.844,166.776,52.291,159.559
C08114=1019.802,37.464,393.860,166.773,52.297,159.559
C08115=1019.797,37.214,393.875,166.771,52.303,159.560
C08116=1019.791,36.964,393.890,166.768,52.309,159.560
C08117=1019.785,36.715,393.905,166.766,52.314,159.561
C08118=1019.780,36.465,393.921,166.764,52.320,159.562
C08119=1019.775,36.216,393.936,166.761,52.326,159.563
C08120=1019.768,35.967,393.951,166.758,52.332,159.563
C08121=1019.763,35.717,393.966,166.756,52.338,159.564
C08122=1019.757,35.468,393.981,166.752,52.345,159.564
C08123=1019.751,35.218,393.996,166.749,52.351,159.565
C08124=1019.745,34.969,394.011,166.747,52.357,159.566
C08125=1019.740,34.719,394.027,166.744,52.363,159.566
C08126=1019.734,34.470,394.041,166.742,52.369,159.567
C08127=1019.728,34.220,394.057,166.739,52.375,159.568
C08128=1019.723,33.971,394.072,166.736,52.381,159.568
C08129=1019.717,33.721,394.087,166.734,52.387,159.569
C08130=1019.712,33.472,394.102,166.731,52.393,159.570
C08131=1019.706,33.223,394.117,166.730,52.399,159.570
C08132=1019.700,32.973,394.132,166.727,52.405,159.571
C08133=1019.695,32.724,394.147,166.724,52.411,159.572
C08134=1019.689,32.474,394.162,166.722,52.417,159.572
C08135=1019.683,32.225,394.177,166.719,52.423,159.573
C08136=1019.678,31.975,394.192,166.717,52.429,159.574
C08137=1019.672,31.726,394.207,166.714,52.435,159.574
C08138=1019.666,31.476,394.222,166.711,52.440,159.575
C08139=1019.660,31.227,394.237,166.708,52.446,159.575
C08140=1019.655,30.977,394.253,166.706,52.452,159.576
C08141=1019.649,30.728,394.267,166.703,52.458,159.577
C08142=1019.644,30.479,394.282,166.701,52.464,159.577
C08143=1019.638,30.229,394.297,166.698,52.470,159.578
C08144=1019.633,29.979,394.312,166.695,52.476,159.578
C08145=1019.627,29.729,394.327,166.693,52.482,159.579
C08146=1019.621,29.480,394.342,166.690,52.488,159.580
C08147=1019.616,29.230,394.357,166.687,52.494,159.580
C08148=1019.610,28.981,394.372,166.685,52.500,159.581
C08149=1019.605,28.732,394.387,166.682,52.506,159.581
C08150=1019.599,28.482,394.402,166.679,52.512,159.582
C08151=1019.594,28.233,394.417,166.676,52.517,159.583
C08152=1019.587,27.983,394.431,166.674,52.523,159.583
C08153=1019.582,27.734,394.447,166.671,52.529,159.584
C08154=1019.577,27.485,394.461,166.669,52.535,159.584
C08155=1019.570,27.201,394.478,166.666,52.542,159.585
C08156=1019.564,26.917,394.495,166.663,52.548,159.586
C08157=1019.557,26.634,394.511,166.660,52.556,159.587
C08158=1019.551,26.351,394.528,166.657,52.562,159.587
C08159=1019.545,26.101,394.543,166.655,52.568,159.588
C08160=1019.540,25.852,394.558,166.652,52.574,159.589
C08161=1019.534,25.601,394.572,166.649,52.580,159.589
C08162=1019.528,25.352,394.587,166.647,52.586,159.590
C08163=1019.523,25.103,394.602,166.644,52.592,159.590
C08164=1019.517,24.853,394.616,166.641,52.598,159.591
C08165=1019.511,24.604,394.631,166.639,52.604,159.592
C08166=1019.505,24.355,394.646,166.636,52.610,159.592
C08167=1019.500,24.104,394.660,166.634,52.616,159.593
C08168=1019.494,23.855,394.675,166.631,52.622,159.594
C08169=1019.488,23.606,394.690,166.628,52.627,159.594
C08170=1019.482,23.356,394.704,166.626,52.634,159.595
C08171=1019.477,23.107,394.719,166.623,52.640,159.595
C08172=1019.472,22.857,394.733,166.620,52.646,159.596
C08173=1019.465,22.608,394.748,166.618,52.652,159.597
C08174=1019.460,22.358,394.763,166.615,52.658,159.597
C08175=1019.455,22.109,394.777,166.612,52.663,159.598
C08176=1019.448,21.859,394.792,166.610,52.669,159.598
C08177=1019.443,21.610,394.806,166.607,52.675,159.599
C08178=1019.438,21.360,394.821,166.605,52.681,159.600
C08179=1019.432,21.111,394.835,166.602,52.687,159.600
C08180=1019.426,20.861,394.850,166.599,52.693,159.601
C08181=1019.420,20.612,394.864,166.596,52.699,159.601
C08182=1019.415,20.362,394.879,166.594,52.705,159.602
C08183=1019.409,20.113,394.894,166.591,52.711,159.603
C08184=1019.404,19.863,394.907,166.589,52.717,159.603
C08185=1019.399,19.614,394.923,166.586,52.722,159.604
C08186=1019.393,19.364,394.936,166.583,52.728,159.604
C08187=1019.387,19.115,394.951,166.581,52.734,159.605
C08188=1019.381,18.865,394.965,166.578,52.741,159.606
C08189=1019.375,18.616,394.980,166.575,52.747,159.606
C08190=1019.370,18.366,394.994,166.572,52.752,159.607
C08191=1019.365,18.116,395.009,166.570,52.758,159.607
C08192=1019.359,17.867,395.023,166.567,52.764,159.608
C08193=1019.353,17.617,395.037,166.565,52.770,159.609
C08194=1019.348,17.368,395.052,166.562,52.776,159.609
C08195=1019.342,17.118,395.066,166.559,52.782,159.610
C08196=1019.336,16.869,395.080,166.557,52.788,159.610
C08197=1019.330,16.620,395.094,166.554,52.794,159.611
C08198=1019.325,16.370,395.108,166.552,52.800,159.612
C08199=1019.319,16.121,395.123,166.549,52.806,159.612
C08200=1019.314,15.870,395.138,166.546,52.811,159.613
C08201=1019.308,15.621,395.151,166.543,52.817,159.613
C08202=1019.302,15.372,395.166,166.541,52.823,159.614
C08203=1019.297,15.122,395.180,166.538,52.830,159.615
C08204=1019.291,14.873,395.194,166.535,52.835,159.615
C08205=1019.285,14.623,395.209,166.533,52.841,159.616
C08206=1019.280,14.374,395.222,166.530,52.847,159.616
C08207=1019.274,14.124,395.236,166.528,52.853,159.617
C08208=1019.268,13.875,395.251,166.525,52.859,159.617
C08209=1019.264,13.625,395.265,166.522,52.865,159.618
C08210=1019.258,13.375,395.280,166.520,52.871,159.619
C08211=1019.252,13.125,395.293,166.517,52.877,159.619
C08212=1019.246,12.877,395.307,166.515,52.883,159.620
C08213=1019.240,12.627,395.321,166.512,52.889,159.620
C08214=1019.235,12.377,395.335,166.509,52.894,159.621
C08215=1019.229,12.128,395.349,166.506,52.900,159.622
C08216=1019.223,11.878,395.363,166.504,52.907,159.622
C08217=1019.218,11.628,395.377,166.500,52.913,159.623
C08218=1019.211,11.379,395.391,166.498,52.919,159.623
C08219=1019.205,11.097,395.407,166.496,52.926,159.624
C08220=1019.199,10.816,395.422,166.492,52.932,159.625
C08221=1019.192,10.533,395.438,166.489,52.939,159.625
C08222=1019.186,10.251,395.454,166.485,52.946,159.626
C08223=1019.180,10.002,395.467,166.483,52.952,159.627
C08224=1019.174,9.753,395.481,166.480,52.958,159.627
C08225=1019.169,9.503,395.495,166.478,52.964,159.628
C08226=1019.163,9.253,395.509,166.475,52.970,159.628
C08227=1019.157,9.003,395.523,166.473,52.976,159.629
C08228=1019.152,8.754,395.537,166.470,52.982,159.630
C08229=1019.145,8.504,395.550,166.467,52.988,159.630
C08230=1019.140,8.255,395.564,166.465,52.994,159.631
C08231=1019.134,8.005,395.578,166.462,53.000,159.631
C08232=1019.129,7.756,395.592,166.460,53.006,159.632
C08233=1019.124,7.506,395.606,166.457,53.012,159.633
C08234=1019.117,7.257,395.619,166.454,53.018,159.633
C08235=1019.112,7.007,395.633,166.452,53.024,159.634
C08236=1019.106,6.758,395.647,166.449,53.030,159.634
C08237=1019.101,6.508,395.661,166.445,53.036,159.635
C08238=1019.095,6.258,395.675,166.442,53.042,159.635
C08239=1019.089,6.009,395.688,166.440,53.048,159.636
C08240=1019.083,5.759,395.702,166.437,53.054,159.637
C08241=1019.078,5.509,395.716,166.434,53.059,159.637
C08242=1019.072,5.260,395.730,166.432,53.066,159.638
C08243=1019.067,5.010,395.744,166.429,53.072,159.638
C08244=1019.061,4.761,395.757,166.427,53.078,159.639
C08245=1019.055,4.511,395.771,166.424,53.083,159.639
C08246=1019.050,4.262,395.785,166.421,53.089,159.640
C08247=1019.044,4.012,395.798,166.419,53.095,159.641
C08248=1019.039,3.763,395.812,166.416,53.101,159.641
C08249=1019.033,3.513,395.826,166.413,53.107,159.642
C08250=1019.027,3.264,395.839,166.411,53.113,159.642
C08251=1019.021,3.014,395.853,166.408,53.119,159.643
C08252=1019.016,2.765,395.867,166.405,53.125,159.643
C08253=1019.010,2.515,395.881,166.403,53.131,159.644
C08254=1019.005,2.265,395.895,166.400,53.137,159.645
C08255=1018.999,2.016,395.907,166.397,53.142,159.645
C08256=1018.994,1.766,395.921,166.395,53.148,159.646
C08257=1018.988,1.516,395.935,166.392,53.154,159.646
C08258=1018.983,1.267,395.949,166.389,53.160,159.647
C08259=1018.977,1.017,395.963,166.387,53.166,159.647
C08260=1018.972,0.769,395.976,166.384,53.171,159.648
C08261=1018.966,0.519,395.990,166.381,53.177,159.648
C08262=1018.961,0.269,396.003,166.379,53.184,159.649
C08263=1018.955,0.019,396.017,166.376,53.189,159.650
C08264=1018.949,-0.230,396.030,166.373,53.195,159.650
C08265=1018.944,-0.479,396.044,166.371,53.201,159.651
C08266=1018.938,-0.729,396.058,166.368,53.207,159.651
C08267=1018.933,-0.979,396.072,166.365,53.213,159.652
C08268=1018.928,-1.229,396.085,166.363,53.218,159.652
C08269=1018.921,-1.478,396.098,166.360,53.224,159.653
C08270=1018.916,-1.728,396.112,166.357,53.230,159.653
C08271=1018.910,-1.977,396.126,166.355,53.236,159.654
C08272=1018.905,-2.227,396.140,166.352,53.241,159.654
C08273=1018.900,-2.476,396.152,166.349,53.247,159.655
C08274=1018.894,-2.726,396.166,166.346,53.253,159.655
C08275=1018.889,-2.975,396.180,166.344,53.259,159.656
C08276=1018.883,-3.225,396.193,166.341,53.265,159.657
C08277=1018.878,-3.475,396.207,166.338,53.271,159.657
C08278=1018.872,-3.724,396.220,166.336,53.277,159.658
C08279=1018.866,-3.974,396.234,166.333,53.282,159.658
C08280=1018.861,-4.224,396.247,166.330,53.288,159.659
C08281=1018.856,-4.473,396.261,166.327,53.294,159.659
C08282=1018.850,-4.723,396.274,166.325,53.300,159.660
C08283=1018.844,-5.003,396.288,166.321,53.306,159.660
C08284=1018.837,-5.283,396.303,166.318,53.313,159.661
C08285=1018.831,-5.563,396.317,166.315,53.320,159.662
C08286=1018.825,-5.842,396.332,166.313,53.327,159.662
C08287=1018.819,-6.092,396.345,166.309,53.333,159.663
C08288=1018.813,-6.342,396.359,166.306,53.339,159.663
C08289=1018.808,-6.592,396.371,166.304,53.345,159.664
C08290=1018.802,-6.841,396.385,166.301,53.351,159.665
C08291=1018.796,-7.091,396.398,166.298,53.357,159.665
C08292=1018.790,-7.340,396.411,166.296,53.363,159.666
C08293=1018.785,-7.590,396.424,166.293,53.369,159.666
C08294=1018.779,-7.839,396.437,166.290,53.374,159.667
C08295=1018.774,-8.089,396.450,166.288,53.380,159.667
C08296=1018.768,-8.338,396.464,166.284,53.387,159.668
C08297=1018.762,-8.588,396.476,166.281,53.392,159.668
C08298=1018.757,-8.838,396.489,166.279,53.398,159.669
C08299=1018.751,-9.087,396.502,166.276,53.405,159.670
C08300=1018.746,-9.337,396.515,166.273,53.410,159.670
C08301=1018.740,-9.587,396.529,166.271,53.416,159.671
C08302=1018.735,-9.837,396.542,166.269,53.422,159.671
C08303=1018.729,-10.085,396.555,166.266,53.428,159.672
C08304=1018.723,-10.335,396.567,166.263,53.434,159.672
C08305=1018.718,-10.585,396.580,166.261,53.440,159.673
C08306=1018.712,-10.835,396.594,166.257,53.446,159.673
C08307=1018.707,-11.084,396.606,166.254,53.452,159.674
C08308=1018.701,-11.333,396.620,166.251,53.458,159.674
C08309=1018.695,-11.583,396.632,166.249,53.464,159.675
C08310=1018.690,-11.834,396.645,166.246,53.470,159.675
C08311=1018.684,-12.082,396.658,166.243,53.475,159.676
C08312=1018.679,-12.332,396.671,166.241,53.481,159.677
C08313=1018.673,-12.582,396.684,166.238,53.487,159.677
C08314=1018.667,-12.831,396.697,166.235,53.493,159.678
C08315=1018.662,-13.081,396.710,166.233,53.499,159.678
C08316=1018.656,-13.331,396.723,166.230,53.505,159.679
C08317=1018.651,-13.580,396.736,166.227,53.511,159.679
C08318=1018.646,-13.830,396.749,166.224,53.517,159.679
C08319=1018.640,-14.079,396.761,166.221,53.523,159.680
C08320=1018.635,-14.330,396.774,166.218,53.528,159.681
C08321=1018.629,-14.578,396.787,166.216,53.534,159.681
C08322=1018.624,-14.828,396.800,166.213,53.540,159.682
C08323=1018.618,-15.078,396.813,166.210,53.546,159.682
C08324=1018.612,-15.327,396.826,166.207,53.551,159.683
C08325=1018.607,-15.577,396.839,166.205,53.558,159.683
C08326=1018.601,-15.827,396.852,166.202,53.563,159.684
C08327=1018.596,-16.076,396.864,166.200,53.569,159.684
C08328=1018.591,-16.326,396.877,166.197,53.575,159.685
C08329=1018.585,-16.576,396.889,166.193,53.581,159.685
C08330=1018.579,-16.825,396.902,166.191,53.587,159.686
C08331=1018.573,-17.075,396.915,166.188,53.594,159.686
C08332=1018.567,-17.324,396.927,166.185,53.599,159.687
C08333=1018.562,-17.574,396.940,166.183,53.605,159.688
C08334=1018.556,-17.824,396.952,166.180,53.611,159.688
C08335=1018.550,-18.073,396.965,166.176,53.617,159.688
C08336=1018.546,-18.323,396.978,166.174,53.623,159.689
C08337=1018.540,-18.573,396.990,166.172,53.630,159.690
C08338=1018.534,-18.823,397.003,166.169,53.635,159.690
C08339=1018.529,-19.072,397.015,166.166,53.641,159.691
C08340=1018.523,-19.322,397.027,166.163,53.647,159.691
C08341=1018.517,-19.571,397.040,166.160,53.653,159.692
C08342=1018.511,-19.821,397.052,166.157,53.659,159.692
C08343=1018.505,-20.071,397.065,166.154,53.665,159.693
C08344=1018.500,-20.320,397.077,166.152,53.671,159.693
C08345=1018.495,-20.570,397.090,166.149,53.677,159.694
C08346=1018.490,-20.819,397.102,166.147,53.683,159.694
C08347=1018.480,-21.237,397.123,166.141,53.693,159.695
C08348=1018.471,-21.656,397.144,166.137,53.703,159.696
C08349=1018.462,-22.074,397.165,166.132,53.713,159.697
C08350=1018.452,-22.493,397.185,166.127,53.722,159.698
C08351=1018.446,-22.743,397.198,166.125,53.729,159.698
C08352=1018.441,-22.992,397.210,166.122,53.734,159.699
C08353=1018.435,-23.242,397.223,166.119,53.740,159.699
C08354=1018.430,-23.491,397.235,166.116,53.746,159.700
C08355=1018.425,-23.741,397.248,166.114,53.752,159.700
C08356=1018.419,-23.990,397.260,166.110,53.758,159.701
C08357=1018.413,-24.240,397.273,166.108,53.764,159.701
C08358=1018.408,-24.489,397.285,166.105,53.770,159.702
C08359=1018.402,-24.739,397.297,166.102,53.776,159.702
C08360=1018.397,-24.988,397.310,166.099,53.781,159.703
C08361=1018.391,-25.239,397.321,166.097,53.787,159.703
C08362=1018.386,-25.488,397.334,166.094,53.793,159.704
C08363=1018.378,-25.847,397.351,166.089,53.802,159.704
C08364=1018.370,-26.206,397.370,166.086,53.810,159.705
C08365=1018.362,-26.565,397.388,166.082,53.818,159.706
C08366=1018.354,-26.925,397.405,166.078,53.827,159.707
C08367=1018.349,-27.174,397.417,166.075,53.833,159.707
C08368=1018.343,-27.424,397.430,166.072,53.839,159.708
C08369=1018.338,-27.673,397.442,166.069,53.844,159.708
C08370=1018.332,-27.924,397.454,166.067,53.851,159.709
C08371=1018.327,-28.173,397.466,166.064,53.856,159.709
C08372=1018.322,-28.422,397.478,166.061,53.863,159.709
C08373=1018.315,-28.672,397.489,166.058,53.869,159.710
C08374=1018.310,-28.922,397.502,166.055,53.874,159.711
C08375=1018.304,-29.172,397.514,166.053,53.881,159.711
C08376=1018.299,-29.421,397.526,166.049,53.886,159.711
C08377=1018.293,-29.671,397.538,166.046,53.893,159.712
C08378=1018.287,-29.921,397.549,166.044,53.899,159.713
C08379=1018.282,-30.170,397.561,166.041,53.904,159.713
C08380=1018.276,-30.420,397.574,166.039,53.911,159.714
C08381=1018.271,-30.670,397.585,166.035,53.916,159.714
C08382=1018.265,-30.919,397.598,166.032,53.923,159.715
C08383=1018.260,-31.169,397.609,166.030,53.928,159.715
C08384=1018.254,-31.418,397.621,166.027,53.934,159.716
C08385=1018.248,-31.668,397.633,166.024,53.940,159.716
C08386=1018.243,-31.918,397.645,166.021,53.946,159.716
C08387=1018.238,-32.167,397.657,166.018,53.952,159.717
C08388=1018.232,-32.417,397.669,166.015,53.958,159.718
C08389=1018.226,-32.666,397.681,166.013,53.964,159.718
C08390=1018.221,-32.917,397.692,166.010,53.970,159.719
C08391=1018.215,-33.166,397.705,166.007,53.976,159.719
C08392=1018.210,-33.416,397.716,166.004,53.982,159.719
C08393=1018.205,-33.666,397.729,166.001,53.988,159.720
C08394=1018.199,-33.915,397.739,165.999,53.994,159.720
C08395=1018.194,-34.164,397.752,165.996,53.999,159.721
C08396=1018.188,-34.415,397.764,165.993,54.005,159.721
C08397=1018.183,-34.664,397.776,165.989,54.011,159.722
C08398=1018.178,-34.914,397.787,165.987,54.018,159.722
C08399=1018.172,-35.163,397.799,165.984,54.023,159.723
C08400=1018.166,-35.413,397.811,165.982,54.029,159.723
C08401=1018.161,-35.662,397.823,165.979,54.035,159.724
C08402=1018.156,-35.912,397.834,165.975,54.041,159.724
C08403=1018.150,-36.162,397.847,165.972,54.047,159.725
C08404=1018.144,-36.412,397.858,165.970,54.053,159.725
C08405=1018.139,-36.661,397.869,165.967,54.059,159.726
C08406=1018.134,-36.911,397.881,165.964,54.064,159.726
C08407=1018.128,-37.188,397.894,165.961,54.071,159.727
C08408=1018.122,-37.466,397.908,165.957,54.077,159.727
C08409=1018.116,-37.743,397.921,165.955,54.084,159.728
C08410=1018.109,-38.020,397.934,165.951,54.090,159.728
C08411=1018.104,-38.270,397.945,165.949,54.096,159.729
C08412=1018.099,-38.520,397.957,165.946,54.102,159.729
C08413=1018.093,-38.769,397.969,165.943,54.109,159.730
C08414=1018.088,-39.019,397.980,165.940,54.114,159.730
C08415=1018.082,-39.269,397.992,165.937,54.120,159.730
C08416=1018.077,-39.518,398.004,165.935,54.126,159.731
C08417=1018.072,-39.768,398.015,165.932,54.131,159.731
C08418=1018.066,-40.017,398.026,165.928,54.138,159.732
C08419=1018.060,-40.268,398.038,165.925,54.143,159.732
C08420=1018.055,-40.517,398.049,165.923,54.150,159.733
C08421=1018.049,-40.767,398.061,165.920,54.155,159.733
C08422=1018.044,-41.016,398.072,165.917,54.162,159.734
C08423=1018.039,-41.266,398.083,165.914,54.168,159.734
C08424=1018.032,-41.516,398.095,165.912,54.174,159.735
C08425=1018.027,-41.766,398.106,165.909,54.180,159.735
C08426=1018.021,-42.015,398.117,165.905,54.186,159.736
C08427=1018.016,-42.265,398.129,165.903,54.192,159.736
C08428=1018.010,-42.514,398.140,165.900,54.198,159.737
C08429=1018.005,-42.765,398.152,165.898,54.204,159.737
C08430=1017.999,-43.014,398.163,165.894,54.210,159.738
C08431=1017.994,-43.264,398.174,165.891,54.215,159.738
C08432=1017.988,-43.513,398.185,165.888,54.221,159.739
C08433=1017.983,-43.763,398.197,165.886,54.227,159.739
C08434=1017.978,-44.013,398.208,165.882,54.234,159.739
C08435=1017.972,-44.262,398.220,165.879,54.239,159.740
C08436=1017.966,-44.512,398.231,165.877,54.245,159.741
C08437=1017.961,-44.762,398.242,165.874,54.251,159.741
C08438=1017.955,-45.011,398.253,165.871,54.258,159.741
C08439=1017.950,-45.261,398.265,165.868,54.263,159.742
C08440=1017.944,-45.511,398.276,165.865,54.269,159.742
C08441=1017.939,-45.760,398.287,165.863,54.275,159.743
C08442=1017.934,-46.010,398.298,165.860,54.280,159.743
C08443=1017.929,-46.260,398.309,165.856,54.287,159.744
C08444=1017.923,-46.509,398.320,165.853,54.293,159.744
C08445=1017.918,-46.759,398.332,165.851,54.298,159.744
C08446=1017.912,-47.008,398.343,165.848,54.304,159.745
C08447=1017.907,-47.259,398.355,165.844,54.310,159.745
C08448=1017.901,-47.508,398.365,165.842,54.317,159.746
C08449=1017.896,-47.758,398.377,165.839,54.322,159.746
C08450=1017.890,-48.008,398.388,165.836,54.328,159.747
C08451=1017.885,-48.258,398.399,165.834,54.334,159.747
C08452=1017.879,-48.507,398.410,165.830,54.340,159.748
C08453=1017.874,-48.757,398.422,165.827,54.345,159.748
C08454=1017.869,-49.006,398.432,165.825,54.352,159.749
C08455=1017.864,-49.256,398.444,165.822,54.357,159.749
C08456=1017.858,-49.506,398.455,165.819,54.363,159.749
C08457=1017.853,-49.755,398.466,165.816,54.369,159.750
C08458=1017.847,-50.005,398.477,165.813,54.375,159.750
C08459=1017.842,-50.255,398.489,165.810,54.380,159.751
C08460=1017.836,-50.504,398.500,165.808,54.387,159.751
C08461=1017.832,-50.755,398.510,165.805,54.392,159.752
C08462=1017.826,-51.004,398.521,165.802,54.398,159.752
C08463=1017.821,-51.254,398.533,165.798,54.404,159.752
C08464=1017.815,-51.503,398.543,165.796,54.410,159.753
C08465=1017.810,-51.753,398.554,165.792,54.417,159.753
C08466=1017.804,-52.003,398.565,165.790,54.423,159.754
C08467=1017.798,-52.252,398.575,165.787,54.428,159.754
C08468=1017.793,-52.503,398.586,165.784,54.435,159.755
C08469=1017.787,-52.752,398.596,165.781,54.441,159.755
C08470=1017.781,-53.002,398.607,165.778,54.447,159.756
C08471=1017.776,-53.279,398.619,165.775,54.454,159.756
C08472=1017.770,-53.557,398.631,165.772,54.460,159.757
C08473=1017.764,-53.834,398.642,165.768,54.467,159.757
C08474=1017.757,-54.112,398.655,165.765,54.474,159.758
C08475=1017.752,-54.362,398.665,165.762,54.480,159.758
C08476=1017.746,-54.611,398.676,165.759,54.487,159.759
C08477=1017.741,-54.861,398.686,165.756,54.492,159.759
C08478=1017.735,-55.111,398.697,165.754,54.498,159.760
C08479=1017.729,-55.360,398.708,165.750,54.504,159.760
C08480=1017.724,-55.610,398.718,165.748,54.511,159.761
C08481=1017.719,-55.859,398.729,165.745,54.516,159.761
C08482=1017.713,-56.109,398.739,165.741,54.523,159.762
C08483=1017.708,-56.359,398.750,165.738,54.528,159.762
C08484=1017.703,-56.609,398.760,165.736,54.535,159.763
C08485=1017.697,-56.859,398.771,165.732,54.541,159.763
C08486=1017.692,-57.109,398.781,165.730,54.547,159.763
C08487=1017.686,-57.358,398.792,165.727,54.553,159.764
C08488=1017.680,-57.608,398.803,165.723,54.558,159.764
C08489=1017.675,-57.857,398.813,165.721,54.565,159.765
C08490=1017.670,-58.107,398.824,165.718,54.570,159.765
C08491=1017.664,-58.357,398.834,165.715,54.577,159.765
C08492=1017.658,-58.606,398.845,165.712,54.583,159.766
C08493=1017.653,-58.856,398.855,165.709,54.589,159.766
C08494=1017.647,-59.106,398.866,165.706,54.595,159.767
C08495=1017.642,-59.356,398.876,165.703,54.601,159.767
C08496=1017.638,-59.606,398.887,165.700,54.607,159.768
C08497=1017.632,-59.855,398.897,165.697,54.613,159.768
C08498=1017.627,-60.105,398.908,165.694,54.619,159.769
C08499=1017.621,-60.355,398.918,165.691,54.625,159.769
C08500=1017.615,-60.605,398.929,165.689,54.631,159.770
C08501=1017.610,-60.854,398.939,165.685,54.637,159.770
C08502=1017.605,-61.104,398.949,165.682,54.642,159.770
C08503=1017.599,-61.354,398.959,165.680,54.649,159.771
C08504=1017.594,-61.603,398.970,165.676,54.655,159.771
C08505=1017.589,-61.853,398.980,165.673,54.660,159.771
C08506=1017.583,-62.102,398.991,165.671,54.666,159.772
C08507=1017.578,-62.352,399.001,165.668,54.672,159.772
C08508=1017.572,-62.603,399.011,165.664,54.678,159.773
C08509=1017.567,-62.851,399.022,165.662,54.684,159.773
C08510=1017.562,-63.101,399.032,165.659,54.690,159.774
C08511=1017.556,-63.352,399.042,165.656,54.695,159.774
C08512=1017.551,-63.601,399.054,165.653,54.702,159.774
C08513=1017.546,-63.851,399.063,165.650,54.708,159.775
C08514=1017.541,-64.101,399.074,165.647,54.713,159.775
C08515=1017.535,-64.350,399.084,165.644,54.720,159.776
C08516=1017.530,-64.600,399.095,165.641,54.726,159.776
C08517=1017.525,-64.850,399.104,165.638,54.731,159.776
C08518=1017.519,-65.099,399.115,165.636,54.737,159.777
C08519=1017.514,-65.349,399.125,165.632,54.743,159.777
C08520=1017.509,-65.599,399.135,165.629,54.749,159.778
C08521=1017.503,-65.848,399.146,165.627,54.755,159.778
C08522=1017.498,-66.098,399.156,165.624,54.761,159.779
C08523=1017.493,-66.348,399.166,165.620,54.767,159.779
C08524=1017.487,-66.598,399.176,165.618,54.773,159.779
C08525=1017.482,-66.847,399.187,165.615,54.778,159.780
C08526=1017.477,-67.097,399.197,165.612,54.784,159.780
C08527=1017.471,-67.347,399.207,165.609,54.790,159.781
C08528=1017.466,-67.597,399.217,165.606,54.796,159.781
C08529=1017.461,-67.846,399.228,165.603,54.802,159.781
C08530=1017.455,-68.096,399.238,165.600,54.807,159.782
C08531=1017.451,-68.345,399.248,165.598,54.814,159.782
C08532=1017.445,-68.595,399.258,165.594,54.819,159.782
C08533=1017.441,-68.846,399.269,165.591,54.825,159.783
C08534=1017.435,-69.095,399.279,165.588,54.831,159.783
C08535=1017.429,-69.373,399.290,165.585,54.837,159.784
C08536=1017.423,-69.652,399.301,165.582,54.844,159.784
C08537=1017.418,-69.931,399.313,165.578,54.850,159.784
C08538=1017.412,-70.209,399.324,165.575,54.856,159.785
C08539=1017.406,-70.459,399.334,165.572,54.862,159.785
C08540=1017.401,-70.709,399.344,165.569,54.869,159.786
C08541=1017.396,-70.959,399.354,165.566,54.874,159.786
C08542=1017.390,-71.209,399.364,165.564,54.880,159.787
C08543=1017.386,-71.458,399.374,165.561,54.886,159.787
C08544=1017.380,-71.709,399.384,165.557,54.892,159.787
C08545=1017.375,-71.958,399.394,165.554,54.897,159.788
C08546=1017.370,-72.208,399.404,165.551,54.903,159.788
C08547=1017.366,-72.457,399.415,165.549,54.908,159.788
C08548=1017.360,-72.707,399.425,165.546,54.914,159.789
C08549=1017.355,-72.957,399.435,165.542,54.921,159.789
C08550=1017.350,-73.207,399.445,165.540,54.926,159.790
C08551=1017.345,-73.456,399.455,165.537,54.932,159.790
C08552=1017.340,-73.706,399.465,165.534,54.937,159.790
C08553=1017.335,-73.956,399.475,165.531,54.943,159.791
C08554=1017.329,-74.206,399.485,165.528,54.949,159.791
C08555=1017.324,-74.455,399.495,165.525,54.955,159.791
C08556=1017.319,-74.705,399.505,165.522,54.960,159.792
C08557=1017.313,-74.954,399.514,165.519,54.966,159.792
C08558=1017.308,-75.205,399.525,165.517,54.972,159.793
C08559=1017.303,-75.455,399.534,165.513,54.978,159.793
C08560=1017.297,-75.704,399.543,165.510,54.984,159.793
C08561=1017.292,-75.954,399.553,165.508,54.990,159.794
C08562=1017.287,-76.204,399.563,165.504,54.996,159.794
C08563=1017.282,-76.453,399.573,165.501,55.002,159.794
C08564=1017.276,-76.703,399.583,165.498,55.007,159.795
C08565=1017.272,-76.953,399.592,165.495,55.014,159.795
C08566=1017.266,-77.203,399.602,165.492,55.020,159.796
C08567=1017.261,-77.452,399.611,165.489,55.025,159.796
C08568=1017.256,-77.702,399.621,165.487,55.031,159.796
C08569=1017.251,-77.952,399.630,165.483,55.038,159.797
C08570=1017.246,-78.202,399.640,165.481,55.043,159.797
C08571=1017.240,-78.452,399.650,165.478,55.049,159.798
C08572=1017.235,-78.701,399.659,165.475,55.055,159.798
C08573=1017.229,-78.951,399.670,165.471,55.061,159.798
C08574=1017.224,-79.201,399.678,165.469,55.067,159.799
C08575=1017.219,-79.450,399.688,165.466,55.073,159.799
C08576=1017.214,-79.700,399.698,165.462,55.079,159.799
C08577=1017.209,-79.950,399.707,165.459,55.084,159.800
C08578=1017.204,-80.200,399.716,165.457,55.090,159.800
C08579=1017.198,-80.450,399.726,165.454,55.095,159.800
C08580=1017.193,-80.699,399.735,165.451,55.102,159.801
C08581=1017.188,-80.949,399.745,165.448,55.108,159.801
C08582=1017.182,-81.199,399.754,165.444,55.115,159.802
C08583=1017.177,-81.449,399.763,165.442,55.120,159.802
C08584=1017.171,-81.698,399.773,165.439,55.126,159.802
C08585=1017.167,-81.948,399.782,165.436,55.133,159.803
C08586=1017.161,-82.198,399.791,165.433,55.138,159.803
C08587=1017.155,-82.448,399.800,165.430,55.144,159.804
C08588=1017.150,-82.697,399.810,165.427,55.151,159.804
C08589=1017.145,-82.947,399.818,165.424,55.156,159.804
C08590=1017.140,-83.197,399.829,165.421,55.162,159.805
C08591=1017.135,-83.447,399.837,165.418,55.169,159.805
C08592=1017.130,-83.696,399.847,165.415,55.174,159.806
C08593=1017.124,-83.947,399.856,165.412,55.180,159.806
C08594=1017.119,-84.197,399.865,165.408,55.186,159.806
C08595=1017.114,-84.446,399.874,165.406,55.192,159.807
C08596=1017.108,-84.696,399.882,165.403,55.198,159.807
C08597=1017.103,-84.946,399.893,165.400,55.204,159.807
C08598=1017.098,-85.195,399.901,165.397,55.210,159.808
C08599=1017.092,-85.476,399.912,165.393,55.216,159.808
C08600=1017.086,-85.757,399.922,165.390,55.223,159.809
C08601=1017.080,-86.037,399.932,165.387,55.230,159.809
C08602=1017.075,-86.318,399.942,165.383,55.237,159.810
C08603=1017.069,-86.567,399.951,165.381,55.242,159.810
C08604=1017.065,-86.817,399.960,165.377,55.249,159.810
C08605=1017.059,-87.067,399.970,165.375,55.255,159.811
C08606=1017.053,-87.317,399.979,165.372,55.260,159.811
C08607=1017.049,-87.567,399.988,165.368,55.266,159.811
C08608=1017.043,-87.816,399.997,165.366,55.273,159.812
C08609=1017.038,-88.067,400.006,165.363,55.278,159.812
C08610=1017.033,-88.316,400.015,165.359,55.284,159.813
C08611=1017.027,-88.565,400.024,165.356,55.290,159.813
C08612=1017.023,-88.815,400.033,165.354,55.296,159.813
C08613=1017.017,-89.065,400.042,165.351,55.301,159.814
C08614=1017.012,-89.315,400.052,165.348,55.308,159.814
C08615=1017.007,-89.565,400.060,165.345,55.314,159.814
C08616=1017.002,-89.815,400.069,165.342,55.319,159.815
C08617=1016.997,-90.064,400.078,165.338,55.325,159.815
C08618=1016.991,-90.314,400.087,165.335,55.331,159.815
C08619=1016.987,-90.564,400.096,165.333,55.337,159.816
C08620=1016.982,-90.814,400.105,165.330,55.343,159.816
C08621=1016.976,-91.064,400.115,165.327,55.349,159.817
C08622=1016.971,-91.313,400.123,165.324,55.355,159.817
C08623=1016.966,-91.563,400.132,165.321,55.360,159.817
C08624=1016.961,-91.813,400.141,165.318,55.366,159.818
C08625=1016.955,-92.062,400.150,165.315,55.372,159.818
C08626=1016.951,-92.312,400.159,165.312,55.378,159.818
C08627=1016.946,-92.562,400.167,165.309,55.383,159.819
C08628=1016.940,-92.812,400.176,165.306,55.389,159.819
C08629=1016.936,-93.062,400.185,165.302,55.395,159.819
C08630=1016.930,-93.312,400.195,165.300,55.402,159.820
C08631=1016.925,-93.562,400.204,165.297,55.407,159.820
C08632=1016.920,-93.811,400.212,165.295,55.413,159.820
///RCONF 1,0,0,0,1,0,0,0,0,0,0,0,0,0,0,0,0,0,0,0,0,0,0,0
C08633=1016.915,-94.061,400.221,165.291,55.419,159.821
C08634=1016.910,-94.311,400.230,165.288,55.425,159.821
C08635=1016.905,-94.561,400.238,165.285,55.430,159.821
C08636=1016.900,-94.810,400.248,165.283,55.436,159.822
C08637=1016.895,-95.060,400.257,165.279,55.442,159.822
C08638=1016.890,-95.310,400.265,165.276,55.448,159.822
C08639=1016.885,-95.560,400.274,165.273,55.453,159.823
C08640=1016.880,-95.809,400.283,165.271,55.459,159.823
C08641=1016.875,-96.059,400.292,165.268,55.465,159.823
C08642=1016.870,-96.309,400.300,165.264,55.471,159.824
C08643=1016.865,-96.559,400.309,165.261,55.476,159.824
C08644=1016.860,-96.809,400.318,165.259,55.482,159.824
C08645=1016.855,-97.059,400.326,165.256,55.488,159.825
C08646=1016.850,-97.308,400.336,165.253,55.493,159.825
C08647=1016.845,-97.558,400.344,165.249,55.499,159.825
C08648=1016.840,-97.807,400.353,165.247,55.505,159.826
C08649=1016.835,-98.058,400.361,165.244,55.511,159.826
C08650=1016.830,-98.308,400.370,165.241,55.516,159.826
C08651=1016.825,-98.557,400.378,165.237,55.522,159.827
C08652=1016.820,-98.807,400.387,165.234,55.528,159.827
C08653=1016.814,-99.057,400.395,165.232,55.534,159.827
C08654=1016.809,-99.307,400.404,165.228,55.541,159.828
C08655=1016.804,-99.556,400.412,165.226,55.546,159.828
C08656=1016.798,-99.806,400.421,165.223,55.552,159.828
C08657=1016.794,-100.056,400.430,165.220,55.558,159.829
C08658=1016.789,-100.306,400.438,165.216,55.564,159.829
C08659=1016.784,-100.556,400.446,165.214,55.569,159.829
C08660=1016.778,-100.806,400.455,165.211,55.576,159.830
C08661=1016.773,-101.056,400.463,165.208,55.582,159.830
C08662=1016.769,-101.305,400.471,165.205,55.587,159.830
C08663=1016.763,-101.588,400.481,165.202,55.594,159.831
C08664=1016.756,-101.871,400.490,165.198,55.600,159.831
C08665=1016.751,-102.153,400.499,165.195,55.607,159.832
C08666=1016.746,-102.436,400.509,165.191,55.614,159.832
C08667=1016.740,-102.686,400.517,165.189,55.620,159.832
C08668=1016.735,-102.936,400.526,165.186,55.625,159.833
C08669=1016.730,-103.185,400.534,165.183,55.631,159.833
C08670=1016.726,-103.435,400.542,165.179,55.637,159.833
C08671=1016.720,-103.685,400.550,165.177,55.643,159.834
C08672=1016.715,-103.934,400.559,165.174,55.648,159.834
C08673=1016.710,-104.185,400.567,165.171,55.654,159.834
C08674=1016.705,-104.434,400.575,165.167,55.660,159.834
C08675=1016.700,-104.684,400.584,165.165,55.666,159.835
C08676=1016.695,-104.934,400.593,165.162,55.672,159.835
C08677=1016.691,-105.184,400.600,165.159,55.677,159.836
C08678=1016.685,-105.434,400.609,165.155,55.683,159.836
C08679=1016.680,-105.683,400.617,165.153,55.689,159.836
C08680=1016.675,-105.934,400.625,165.150,55.695,159.836
C08681=1016.670,-106.183,400.633,165.148,55.701,159.837
C08682=1016.666,-106.433,400.641,165.144,55.707,159.837
C08683=1016.660,-106.683,400.649,165.141,55.713,159.838
C08684=1016.655,-106.932,400.658,165.138,55.719,159.838
C08685=1016.650,-107.183,400.665,165.136,55.724,159.838
C08686=1016.645,-107.432,400.674,165.133,55.730,159.839
C08687=1016.640,-107.681,400.682,165.129,55.736,159.839
C08688=1016.635,-107.932,400.690,165.126,55.742,159.839
C08689=1016.630,-108.181,400.698,165.124,55.748,159.840
C08690=1016.625,-108.432,400.706,165.121,55.753,159.840
C08691=1016.620,-108.681,400.714,165.117,55.759,159.840
C08692=1016.615,-108.931,400.722,165.115,55.765,159.840
C08693=1016.609,-109.181,400.730,165.112,55.771,159.841
C08694=1016.604,-109.431,400.738,165.108,55.777,159.841
C08695=1016.600,-109.681,400.745,165.105,55.782,159.841
C08696=1016.595,-109.930,400.753,165.103,55.788,159.842
C08697=1016.590,-110.181,400.761,165.100,55.794,159.842
C08698=1016.585,-110.430,400.769,165.096,55.800,159.842
C08699=1016.580,-110.680,400.777,165.093,55.806,159.843
C08700=1016.575,-110.930,400.786,165.091,55.812,159.843
C08701=1016.570,-111.180,400.793,165.088,55.818,159.844
C08702=1016.565,-111.429,400.801,165.085,55.824,159.844
C08703=1016.560,-111.679,400.809,165.082,55.830,159.844
C08704=1016.555,-111.929,400.816,165.079,55.835,159.844
C08705=1016.550,-112.178,400.825,165.077,55.841,159.845
C08706=1016.545,-112.429,400.832,165.074,55.847,159.845
C08707=1016.540,-112.678,400.841,165.070,55.853,159.845
C08708=1016.535,-112.928,400.848,165.067,55.859,159.846
C08709=1016.530,-113.178,400.856,165.065,55.864,159.846
C08710=1016.525,-113.427,400.864,165.062,55.870,159.846
C08711=1016.520,-113.677,400.871,165.059,55.875,159.846
C08712=1016.515,-113.928,400.879,165.055,55.881,159.847
C08713=1016.510,-114.177,400.887,165.052,55.887,159.847
C08714=1016.506,-114.427,400.895,165.049,55.892,159.847
C08715=1016.501,-114.677,400.903,165.047,55.898,159.848
C08716=1016.496,-114.926,400.911,165.044,55.904,159.848
C08717=1016.490,-115.176,400.918,165.040,55.910,159.848
C08718=1016.486,-115.426,400.925,165.038,55.916,159.849
C08719=1016.481,-115.676,400.933,165.035,55.921,159.849
C08720=1016.476,-115.927,400.941,165.032,55.927,159.849
C08721=1016.471,-116.175,400.948,165.028,55.933,159.849
C08722=1016.466,-116.426,400.956,165.026,55.939,159.850
C08723=1016.461,-116.675,400.964,165.023,55.945,159.850
C08724=1016.456,-116.926,400.971,165.020,55.950,159.851
C08725=1016.451,-117.175,400.978,165.018,55.956,159.851
C08726=1016.446,-117.425,400.987,165.014,55.962,159.851
C08727=1016.440,-117.708,400.995,165.011,55.969,159.851
C08728=1016.435,-117.991,401.004,165.008,55.976,159.852
C08729=1016.430,-118.273,401.012,165.005,55.982,159.852
C08730=1016.424,-118.556,401.021,165.001,55.988,159.853
C08731=1016.419,-118.807,401.028,164.999,55.994,159.853
C08732=1016.414,-119.056,401.036,164.995,56.000,159.853
C08733=1016.409,-119.306,401.043,164.992,56.006,159.854
C08734=1016.404,-119.555,401.051,164.989,56.012,159.854
C08735=1016.399,-119.806,401.059,164.987,56.018,159.854
C08736=1016.394,-120.055,401.066,164.984,56.023,159.855
C08737=1016.389,-120.305,401.073,164.980,56.029,159.855
C08738=1016.385,-120.555,401.081,164.978,56.035,159.855
C08739=1016.379,-120.805,401.088,164.974,56.040,159.855
C08740=1016.375,-121.055,401.095,164.972,56.046,159.856
C08741=1016.370,-121.304,401.103,164.969,56.052,159.856
C08742=1016.365,-121.554,401.110,164.966,56.057,159.856
C08743=1016.360,-121.804,401.117,164.963,56.063,159.856
C08744=1016.355,-122.054,401.125,164.960,56.069,159.857
C08745=1016.350,-122.304,401.132,164.957,56.075,159.857
C08746=1016.345,-122.554,401.140,164.954,56.081,159.857
C08747=1016.341,-122.804,401.147,164.952,56.086,159.858
C08748=1016.335,-123.054,401.154,164.949,56.092,159.858
C08749=1016.331,-123.303,401.162,164.945,56.098,159.858
C08750=1016.326,-123.553,401.169,164.943,56.104,159.859
C08751=1016.321,-123.803,401.176,164.939,56.109,159.859
C08752=1016.316,-124.052,401.184,164.937,56.115,159.859
C08753=1016.311,-124.303,401.191,164.934,56.120,159.859
C08754=1016.306,-124.552,401.198,164.931,56.126,159.860
C08755=1016.302,-124.802,401.205,164.929,56.132,159.860
C08756=1016.297,-125.052,401.212,164.925,56.138,159.860
C08757=1016.292,-125.302,401.219,164.922,56.144,159.861
C08758=1016.287,-125.552,401.227,164.919,56.149,159.861
C08759=1016.282,-125.802,401.234,164.917,56.155,159.861
C08760=1016.277,-126.051,401.241,164.914,56.161,159.862
C08761=1016.272,-126.302,401.248,164.910,56.167,159.862
C08762=1016.267,-126.551,401.255,164.908,56.173,159.862
C08763=1016.263,-126.801,401.262,164.905,56.178,159.863
C08764=1016.257,-127.051,401.269,164.902,56.183,159.863
C08765=1016.253,-127.301,401.277,164.899,56.189,159.863
C08766=1016.248,-127.551,401.283,164.896,56.195,159.863
C08767=1016.244,-127.800,401.290,164.894,56.201,159.864
C08768=1016.239,-128.049,401.297,164.890,56.207,159.864
C08769=1016.234,-128.300,401.305,164.887,56.213,159.864
C08770=1016.229,-128.549,401.313,164.885,56.217,159.865
C08771=1016.225,-128.799,401.321,164.882,56.221,159.865
C08772=1016.222,-129.048,401.330,164.880,56.225,159.865
C08773=1016.219,-129.298,401.339,164.877,56.228,159.864
C08774=1016.216,-129.547,401.350,164.874,56.231,159.864
C08775=1016.214,-129.797,401.361,164.872,56.233,159.864
C08776=1016.212,-130.047,401.373,164.869,56.235,159.864
C08777=1016.211,-130.297,401.384,164.867,56.235,159.863
C08778=1016.209,-130.546,401.397,164.864,56.236,159.863
C08779=1016.209,-130.796,401.410,164.862,56.236,159.862
C08780=1016.208,-131.045,401.424,164.859,56.234,159.861
C08781=1016.209,-131.295,401.439,164.857,56.233,159.860
C08782=1016.209,-131.545,401.454,164.856,56.231,159.860
C08783=1016.209,-131.795,401.469,164.854,56.229,159.859
C08784=1016.210,-132.045,401.486,164.852,56.226,159.858
C08785=1016.212,-132.294,401.503,164.849,56.222,159.856
C08786=1016.214,-132.543,401.520,164.848,56.218,159.855
C08787=1016.217,-132.793,401.538,164.846,56.213,159.854
C08788=1016.220,-133.043,401.556,164.844,56.208,159.853
C08789=1016.222,-133.292,401.576,164.843,56.202,159.851
C08790=1016.225,-133.542,401.595,164.841,56.196,159.850
C08791=1015.975,-133.568,401.202,164.804,56.563,159.905
C08792=1015.972,-133.319,401.182,164.806,56.569,159.907
C08793=1015.969,-133.069,401.162,164.807,56.576,159.908
C08794=1015.966,-132.819,401.143,164.808,56.581,159.910
C08795=1015.964,-132.570,401.125,164.811,56.586,159.911
C08796=1015.962,-132.320,401.108,164.812,56.590,159.912
C08797=1015.960,-132.071,401.091,164.815,56.594,159.914
C08798=1015.959,-131.821,401.075,164.817,56.597,159.915
C08799=1015.958,-131.571,401.059,164.819,56.599,159.916
C08800=1015.958,-131.321,401.044,164.821,56.601,159.916
C08801=1015.958,-131.071,401.030,164.823,56.602,159.917
C08802=1015.959,-130.822,401.015,164.825,56.603,159.918
C08803=1015.960,-130.573,401.002,164.828,56.603,159.919
C08804=1015.960,-130.322,400.990,164.830,56.602,159.919
C08805=1015.962,-130.073,400.977,164.832,56.601,159.919
C08806=1015.964,-129.823,400.966,164.835,56.600,159.920
C08807=1015.966,-129.574,400.955,164.838,56.598,159.920
C08808=1015.968,-129.324,400.945,164.840,56.596,159.920
C08809=1015.972,-129.075,400.935,164.843,56.592,159.921
C08810=1015.975,-128.825,400.926,164.846,56.589,159.921
C08811=1015.978,-128.575,400.918,164.848,56.584,159.920
C08812=1015.983,-128.326,400.910,164.850,56.579,159.920
C08813=1015.987,-128.076,400.902,164.853,56.574,159.920
C08814=1015.993,-127.827,400.895,164.857,56.568,159.920
C08815=1015.997,-127.577,400.889,164.859,56.562,159.919
C08816=1016.002,-127.327,400.882,164.862,56.556,159.919
C08817=1016.007,-127.077,400.874,164.865,56.551,159.919
C08818=1016.012,-126.828,400.867,164.867,56.545,159.918
C08819=1016.016,-126.577,400.860,164.871,56.539,159.918
C08820=1016.021,-126.328,400.853,164.874,56.533,159.918
C08821=1016.026,-126.078,400.846,164.876,56.527,159.918
C08822=1016.032,-125.828,400.839,164.879,56.521,159.917
C08823=1016.036,-125.578,400.832,164.882,56.516,159.917
C08824=1016.041,-125.328,400.825,164.885,56.510,159.917
C08825=1016.046,-125.078,400.818,164.888,56.504,159.916
C08826=1016.051,-124.829,400.811,164.891,56.498,159.916
C08827=1016.055,-124.579,400.803,164.893,56.492,159.916
C08828=1016.061,-124.329,400.796,164.896,56.486,159.915
C08829=1016.065,-124.079,400.790,164.900,56.480,159.915
C08830=1016.069,-123.829,400.782,164.903,56.475,159.915
C08831=1016.075,-123.579,400.775,164.905,56.469,159.915
C08832=1016.079,-123.330,400.768,164.908,56.464,159.914
C08833=1016.084,-123.079,400.760,164.911,56.458,159.914
C08834=1016.089,-122.830,400.753,164.914,56.452,159.914
C08835=1016.094,-122.580,400.746,164.917,56.446,159.913
C08836=1016.099,-122.330,400.738,164.920,56.440,159.913
C08837=1016.104,-122.081,400.731,164.922,56.434,159.913
C08838=1016.109,-121.830,400.723,164.925,56.429,159.912
C08839=1016.114,-121.581,400.716,164.929,56.423,159.912
C08840=1016.118,-121.331,400.709,164.931,56.417,159.912
C08841=1016.123,-121.081,400.701,164.934,56.411,159.911
C08842=1016.127,-120.831,400.694,164.937,56.405,159.911
C08843=1016.133,-120.581,400.687,164.939,56.400,159.911
C08844=1016.138,-120.332,400.679,164.943,56.393,159.911
C08845=1016.142,-120.081,400.672,164.946,56.388,159.910
C08846=1016.148,-119.832,400.665,164.948,56.382,159.910
C08847=1016.153,-119.582,400.657,164.951,56.376,159.909
C08848=1016.157,-119.332,400.650,164.955,56.370,159.909
C08849=1016.162,-119.083,400.643,164.957,56.364,159.909
C08850=1016.167,-118.832,400.635,164.960,56.358,159.909
C08851=1016.171,-118.583,400.628,164.963,56.353,159.908
C08852=1016.177,-118.300,400.619,164.966,56.347,159.908
C08853=1016.183,-118.017,400.610,164.970,56.340,159.908
C08854=1016.188,-117.735,400.603,164.973,56.333,159.907
C08855=1016.194,-117.452,400.593,164.976,56.326,159.907
C08856=1016.199,-117.203,400.586,164.979,56.320,159.906
C08857=1016.204,-116.952,400.578,164.982,56.314,159.906
C08858=1016.209,-116.702,400.571,164.985,56.308,159.906
C08859=1016.213,-116.452,400.563,164.988,56.302,159.905
C08860=1016.219,-116.202,400.556,164.990,56.297,159.905
C08861=1016.223,-115.953,400.548,164.994,56.290,159.905
C08862=1016.228,-115.703,400.540,164.997,56.285,159.905
C08863=1016.233,-115.453,400.533,164.999,56.279,159.904
C08864=1016.238,-115.203,400.526,165.002,56.273,159.904
C08865=1016.243,-114.954,400.518,165.006,56.267,159.904
C08866=1016.248,-114.704,400.510,165.008,56.261,159.903
C08867=1016.253,-114.454,400.502,165.011,56.256,159.903
C08868=1016.257,-114.204,400.495,165.014,56.250,159.903
C08869=1016.263,-113.954,400.487,165.017,56.244,159.902
C08870=1016.268,-113.705,400.479,165.020,56.238,159.902
C08871=1016.273,-113.455,400.472,165.023,56.232,159.902
C08872=1016.278,-113.204,400.464,165.025,56.227,159.901
C08873=1016.282,-112.955,400.456,165.029,56.220,159.901
C08874=1016.287,-112.705,400.448,165.032,56.215,159.901
C08875=1016.292,-112.455,400.440,165.035,56.209,159.900
C08876=1016.297,-112.206,400.432,165.038,56.203,159.900
C08877=1016.303,-111.956,400.425,165.041,56.197,159.900
C08878=1016.307,-111.706,400.417,165.044,56.191,159.900
C08879=1016.312,-111.456,400.409,165.046,56.186,159.899
C08880=1016.317,-111.206,400.401,165.049,56.179,159.899
C08881=1016.322,-110.957,400.393,165.052,56.173,159.898
C08882=1016.327,-110.706,400.385,165.055,56.167,159.898
C08883=1016.332,-110.456,400.378,165.059,56.161,159.898
C08884=1016.336,-110.207,400.369,165.061,56.155,159.897
C08885=1016.342,-109.957,400.362,165.064,56.150,159.897
C08886=1016.347,-109.707,400.354,165.067,56.144,159.897
C08887=1016.352,-109.458,400.346,165.070,56.138,159.897
C08888=1016.357,-109.207,400.339,165.073,56.132,159.896
C08889=1016.362,-108.958,400.330,165.075,56.126,159.896
C08890=1016.366,-108.708,400.323,165.079,56.119,159.895
C08891=1016.372,-108.458,400.314,165.081,56.114,159.895
C08892=1016.377,-108.208,400.306,165.084,56.108,159.895
C08893=1016.382,-107.958,400.298,165.088,56.102,159.895
C08894=1016.386,-107.709,400.291,165.091,56.096,159.894
C08895=1016.391,-107.459,400.282,165.093,56.090,159.894
C08896=1016.396,-107.209,400.274,165.097,56.084,159.894
C08897=1016.402,-106.959,400.266,165.100,56.078,159.893
C08898=1016.406,-106.709,400.258,165.102,56.072,159.893
C08899=1016.411,-106.460,400.250,165.105,56.066,159.892
C08900=1016.417,-106.210,400.241,165.108,56.060,159.892
C08901=1016.422,-105.960,400.234,165.111,56.054,159.892
C08902=1016.426,-105.711,400.226,165.114,56.049,159.891
C08903=1016.431,-105.460,400.218,165.117,56.043,159.891
C08904=1016.436,-105.210,400.209,165.120,56.037,159.891
C08905=1016.442,-104.961,400.201,165.123,56.031,159.890
C08906=1016.447,-104.710,400.193,165.126,56.025,159.890
C08907=1016.451,-104.461,400.185,165.129,56.019,159.890
C08908=1016.457,-104.212,400.176,165.131,56.013,159.889
C08909=1016.462,-103.961,400.169,165.134,56.007,159.889
C08910=1016.467,-103.712,400.160,165.138,56.001,159.889
C08911=1016.472,-103.462,400.152,165.140,55.995,159.888
C08912=1016.476,-103.212,400.144,165.143,55.990,159.888
C08913=1016.481,-102.962,400.135,165.147,55.983,159.888
C08914=1016.486,-102.713,400.127,165.150,55.978,159.887
C08915=1016.491,-102.463,400.118,165.152,55.972,159.887
C08916=1016.498,-102.180,400.109,165.155,55.965,159.887
C08917=1016.503,-101.898,400.100,165.159,55.958,159.886
C08918=1016.508,-101.615,400.090,165.162,55.952,159.886
C08919=1016.514,-101.332,400.081,165.165,55.945,159.885
C08920=1016.520,-101.082,400.073,165.169,55.939,159.885
C08921=1016.524,-100.832,400.064,165.172,55.933,159.885
C08922=1016.529,-100.583,400.056,165.174,55.927,159.884
C08923=1016.534,-100.333,400.048,165.178,55.920,159.884
C08924=1016.539,-100.083,400.039,165.180,55.915,159.884
C08925=1016.544,-99.834,400.031,165.184,55.908,159.883
C08926=1016.550,-99.584,400.022,165.187,55.903,159.883
C08927=1016.555,-99.334,400.014,165.189,55.897,159.883
C08928=1016.560,-99.085,400.005,165.193,55.890,159.882
C08929=1016.565,-98.834,399.998,165.195,55.885,159.882
C08930=1016.570,-98.584,399.989,165.198,55.879,159.881
C08931=1016.575,-98.334,399.980,165.202,55.873,159.881
C08932=1016.580,-98.085,399.972,165.204,55.866,159.881
C08933=1016.585,-97.835,399.963,165.207,55.861,159.880
C08934=1016.591,-97.585,399.955,165.210,55.854,159.880
C08935=1016.595,-97.335,399.946,165.213,55.849,159.880
C08936=1016.600,-97.086,399.937,165.216,55.843,159.879
C08937=1016.605,-96.836,399.928,165.218,55.837,159.879
C08938=1016.610,-96.586,399.920,165.222,55.831,159.879
C08939=1016.616,-96.336,399.911,165.225,55.826,159.878
C08940=1016.620,-96.086,399.902,165.228,55.820,159.878
C08941=1016.625,-95.837,399.894,165.231,55.814,159.878
C08942=1016.629,-95.587,399.885,165.234,55.808,159.877
C08943=1016.634,-95.337,399.876,165.237,55.802,159.877
C08944=1016.640,-95.088,399.868,165.239,55.796,159.876
C08945=1016.645,-94.837,399.858,165.243,55.790,159.876
C08946=1016.650,-94.587,399.850,165.245,55.784,159.876
C08947=1016.656,-94.338,399.841,165.248,55.778,159.876
C08948=1016.660,-94.088,399.832,165.252,55.772,159.875
C08949=1016.666,-93.838,399.823,165.255,55.767,159.875
C08950=1016.670,-93.588,399.814,165.257,55.761,159.875
C08951=1016.675,-93.339,399.806,165.260,55.755,159.874
C08952=1016.681,-93.089,399.797,165.263,55.748,159.874
C08953=1016.685,-92.839,399.788,165.266,55.743,159.873
C08954=1016.691,-92.590,399.779,165.269,55.737,159.873
C08955=1016.695,-92.340,399.770,165.272,55.731,159.873
///RCONF 1,0,0,0,0,0,0,0,0,0,0,0,0,0,0,0,0,0,0,0,0,0,0,0
C08956=1016.700,-92.090,399.761,165.275,55.725,159.872
C08957=1016.706,-91.840,399.753,165.278,55.720,159.872
C08958=1016.710,-91.590,399.744,165.281,55.713,159.872
C08959=1016.716,-91.341,399.735,165.284,55.707,159.871
C08960=1016.720,-91.091,399.725,165.287,55.701,159.871
C08961=1016.726,-90.841,399.717,165.290,55.695,159.871
C08962=1016.731,-90.591,399.708,165.293,55.689,159.870
C08963=1016.736,-90.341,399.699,165.295,55.683,159.870
C08964=1016.742,-90.092,399.690,165.299,55.677,159.870
C08965=1016.746,-89.842,399.681,165.302,55.671,159.869
C08966=1016.751,-89.592,399.672,165.304,55.666,159.869
C08967=1016.756,-89.342,399.663,165.308,55.659,159.868
C08968=1016.761,-89.093,399.654,165.310,55.653,159.868
C08969=1016.767,-88.843,399.645,165.313,55.648,159.868
C08970=1016.772,-88.593,399.636,165.316,55.641,159.867
C08971=1016.777,-88.343,399.627,165.319,55.635,159.867
C08972=1016.782,-88.093,399.618,165.323,55.629,159.867
C08973=1016.787,-87.844,399.609,165.326,55.623,159.866
C08974=1016.792,-87.594,399.601,165.328,55.617,159.866
C08975=1016.797,-87.345,399.591,165.332,55.611,159.865
C08976=1016.803,-87.094,399.582,165.334,55.605,159.865
C08977=1016.808,-86.844,399.573,165.338,55.598,159.864
C08978=1016.813,-86.595,399.564,165.340,55.593,159.864
C08979=1016.818,-86.345,399.555,165.343,55.587,159.864
C08980=1016.824,-86.064,399.545,165.346,55.580,159.863
C08981=1016.830,-85.784,399.535,165.350,55.573,159.863
C08982=1016.836,-85.503,399.525,165.353,55.567,159.862
C08983=1016.842,-85.223,399.514,165.357,55.559,159.862
C08984=1016.847,-84.973,399.505,165.359,55.553,159.861
C08985=1016.852,-84.723,399.496,165.362,55.547,159.861
C08986=1016.857,-84.474,399.487,165.366,55.541,159.861
C08987=1016.862,-84.224,399.477,165.368,55.535,159.860
C08988=1016.868,-83.974,399.469,165.372,55.529,159.860
C08989=1016.873,-83.725,399.460,165.374,55.522,159.859
C08990=1016.878,-83.474,399.450,165.377,55.517,159.859
C08991=1016.884,-83.225,399.441,165.381,55.511,159.859
C08992=1016.888,-82.975,399.432,165.383,55.504,159.858
C08993=1016.894,-82.726,399.423,165.387,55.498,159.858
C08994=1016.899,-82.475,399.413,165.389,55.492,159.857
C08995=1016.904,-82.225,399.405,165.393,55.486,159.857
C08996=1016.910,-81.976,399.395,165.395,55.480,159.857
C08997=1016.915,-81.726,399.386,165.399,55.473,159.856
C08998=1016.921,-81.477,399.377,165.401,55.468,159.856
C08999=1016.925,-81.226,399.368,165.404,55.461,159.855
C09000=1016.931,-80.977,399.358,165.407,55.455,159.855
C09001=1016.936,-80.727,399.349,165.410,55.449,159.855
C09002=1016.941,-80.478,399.340,165.413,55.443,159.854
C09003=1016.947,-80.227,399.330,165.416,55.436,159.854
C09004=1016.952,-79.978,399.321,165.419,55.430,159.853
C09005=1016.957,-79.728,399.311,165.422,55.425,159.853
C09006=1016.962,-79.478,399.301,165.425,55.419,159.853
C09007=1016.968,-79.228,399.293,165.428,55.412,159.852
C09008=1016.972,-78.979,399.283,165.431,55.407,159.852
C09009=1016.978,-78.729,399.273,165.434,55.401,159.852
C09010=1016.982,-78.479,399.264,165.437,55.394,159.851
C09011=1016.988,-78.230,399.255,165.440,55.389,159.851
C09012=1016.993,-77.980,399.244,165.442,55.383,159.850
C09013=1016.998,-77.730,399.235,165.446,55.377,159.850
C09014=1017.004,-77.480,399.226,165.448,55.370,159.849
C09015=1017.009,-77.231,399.216,165.451,55.365,159.849
C09016=1017.014,-76.981,399.206,165.455,55.359,159.849
C09017=1017.019,-76.731,399.196,165.457,55.352,159.848
C09018=1017.024,-76.481,399.188,165.461,55.346,159.848
C09019=1017.030,-76.231,399.177,165.463,55.340,159.847
C09020=1017.035,-75.982,399.168,165.466,55.334,159.847
C09021=1017.040,-75.733,399.158,165.470,55.328,159.847
C09022=1017.045,-75.482,399.149,165.472,55.322,159.846
C09023=1017.050,-75.233,399.139,165.475,55.316,159.846
C09024=1017.056,-74.982,399.129,165.479,55.310,159.846
C09025=1017.061,-74.733,399.120,165.481,55.304,159.845
C09026=1017.067,-74.483,399.110,165.485,55.298,159.845
C09027=1017.072,-74.234,399.100,165.487,55.292,159.844
C09028=1017.077,-73.984,399.090,165.490,55.287,159.844
C09029=1017.082,-73.734,399.080,165.492,55.280,159.843
C09030=1017.087,-73.484,399.070,165.496,55.274,159.843
C09031=1017.092,-73.235,399.060,165.499,55.269,159.843
C09032=1017.098,-72.985,399.050,165.502,55.263,159.842
C09033=1017.102,-72.735,399.040,165.504,55.257,159.842
C09034=1017.108,-72.485,399.030,165.508,55.250,159.842
C09035=1017.113,-72.236,399.020,165.511,55.245,159.841
C09036=1017.118,-71.986,399.010,165.513,55.239,159.841
C09037=1017.123,-71.736,399.000,165.516,55.234,159.840
C09038=1017.128,-71.486,398.990,165.519,55.227,159.840
C09039=1017.133,-71.237,398.980,165.522,55.221,159.840
C09040=1017.139,-70.987,398.970,165.525,55.216,159.839
C09041=1017.143,-70.737,398.960,165.529,55.210,159.839
C09042=1017.148,-70.487,398.949,165.531,55.204,159.839
C09043=1017.153,-70.237,398.940,165.534,55.198,159.838
C09044=1017.159,-69.959,398.928,165.537,55.191,159.837
C09045=1017.165,-69.680,398.917,165.540,55.184,159.837
C09046=1017.171,-69.402,398.905,165.544,55.178,159.837
C09047=1017.177,-69.123,398.894,165.547,55.171,159.836
C09048=1017.182,-68.874,398.884,165.550,55.165,159.836
C09049=1017.187,-68.624,398.874,165.552,55.159,159.835
C09050=1017.192,-68.374,398.864,165.556,55.153,159.835
C09051=1017.198,-68.124,398.854,165.559,55.147,159.834
C09052=1017.203,-67.874,398.844,165.561,55.141,159.834
C09053=1017.208,-67.625,398.833,165.565,55.135,159.834
C09054=1017.214,-67.375,398.823,165.567,55.129,159.833
C09055=1017.218,-67.126,398.813,165.570,55.123,159.833
C09056=1017.224,-66.876,398.803,165.574,55.117,159.833
C09057=1017.229,-66.626,398.793,165.576,55.111,159.832
C09058=1017.233,-66.376,398.783,165.579,55.105,159.832
C09059=1017.239,-66.127,398.772,165.583,55.099,159.831
C09060=1017.245,-65.876,398.762,165.585,55.093,159.831
C09061=1017.249,-65.627,398.752,165.588,55.087,159.830
C09062=1017.255,-65.377,398.742,165.592,55.081,159.830
C09063=1017.261,-65.127,398.731,165.594,55.075,159.829
C09064=1017.265,-64.878,398.721,165.597,55.069,159.829
C09065=1017.271,-64.628,398.711,165.600,55.063,159.829
C09066=1017.276,-64.378,398.701,165.603,55.057,159.828
C09067=1017.281,-64.129,398.690,165.606,55.051,159.828
C09068=1017.287,-63.879,398.680,165.609,55.045,159.827
C09069=1017.292,-63.629,398.670,165.612,55.039,159.827
C09070=1017.297,-63.380,398.659,165.614,55.033,159.826
C09071=1017.303,-63.130,398.649,165.618,55.027,159.826
C09072=1017.308,-62.880,398.639,165.620,55.020,159.826
C09073=1017.313,-62.631,398.629,165.624,55.014,159.825
C09074=1017.319,-62.381,398.618,165.627,55.009,159.825
C09075=1017.324,-62.131,398.608,165.629,55.002,159.824
C09076=1017.330,-61.881,398.597,165.633,54.996,159.824
C09077=1017.335,-61.632,398.588,165.635,54.990,159.823
C09078=1017.340,-61.381,398.577,165.638,54.984,159.823
C09079=1017.345,-61.132,398.566,165.641,54.978,159.823
C09080=1017.351,-60.882,398.556,165.644,54.972,159.822
C09081=1017.356,-60.632,398.546,165.647,54.965,159.822
C09082=1017.361,-60.383,398.535,165.650,54.960,159.821
C09083=1017.367,-60.133,398.525,165.652,54.953,159.821
C09084=1017.372,-59.883,398.514,165.656,54.947,159.820
C09085=1017.377,-59.634,398.504,165.658,54.941,159.820
C09086=1017.383,-59.384,398.494,165.662,54.935,159.820
C09087=1017.388,-59.134,398.483,165.665,54.929,159.819
C09088=1017.394,-58.884,398.473,165.667,54.922,159.818
C09089=1017.400,-58.635,398.462,165.671,54.916,159.818
C09090=1017.404,-58.385,398.452,165.673,54.910,159.817
C09091=1017.410,-58.136,398.442,165.677,54.904,159.817
C09092=1017.416,-57.886,398.431,165.679,54.898,159.817
C09093=1017.421,-57.636,398.420,165.682,54.892,159.816
C09094=1017.426,-57.386,398.410,165.685,54.886,159.816
C09095=1017.431,-57.136,398.400,165.688,54.879,159.815
C09096=1017.437,-56.887,398.389,165.691,54.873,159.815
C09097=1017.442,-56.637,398.379,165.694,54.867,159.814
C09098=1017.448,-56.387,398.368,165.696,54.861,159.814
C09099=1017.453,-56.137,398.358,165.700,54.855,159.813
